THIS^.testLsbIsNotEqualTo(
	valueToTest := THIS^.LSB_ONLY,
	unexpectedValue := TRUE
);	
THIS^.testLsbIsNotEqualTo(
	valueToTest := THIS^.LSB_ONLY,
	unexpectedValue := FALSE
);
THIS^.testLsbIsNotEqualTo(
	valueToTest := THIS^.MSB_ONLY,
	unexpectedValue := TRUE
);	
THIS^.testLsbIsNotEqualTo(
	valueToTest := THIS^.MSB_ONLY,
	unexpectedValue := FALSE
);

TcUnit.TEST_FINISHED();
END_METHOD

(*

simple summary
==================
This test method tests ``assert.bitNumber.simple.lsbIsSet``
of CNM_AssertionInterfaces library with various inputs

.. <legal notes>

legal notes
=================
| SPDX-FileCopyrightText: © 2022 ekvip automation GmbH <info@ekvip.de>
| SPDX-License-Identifier: Apache-2.0
| For details check: Apache-2.0_

.. _Apache-2.0: https://www.apache.org/licenses/LICENSE-2.0

.. </legal notes>

*)

METHOD runLsbIsSetTests
VAR
	(* it's just part of the test data *)
	valueToTest	:WORD;
	(* multiplier to get various bit patterns *)
	multiplier	:UINT;
END_VAR
RETURN (NOT TcUnit.TEST_ORDERED(THIS^.getTestNameFor('lsbIsSet')));

FOR multiplier := THIS^.FIRST_MULTIPLIER TO THIS^.LAST_MULTIPLIER DO
	valueToTest := (THIS^.MULTIPLICAND * multiplier);
	THIS^.testLsbIsSet(
		valueToTest := valueToTest
	);
END_FOR

THIS^.testLsbIsSet(
	valueToTest := THIS^.MSB_ONLY
);	
THIS^.testLsbIsSet(
	valueToTest := THIS^.MSB_ONLY
);

TcUnit.TEST_FINISHED();
END_METHOD

(*

simple summary
==================
This test method tests ``assert.bitNumber.simple.lsbIsUnset``
of CNM_AssertionInterfaces library with various inputs

.. <legal notes>

legal notes
=================
| SPDX-FileCopyrightText: © 2022 ekvip automation GmbH <info@ekvip.de>
| SPDX-License-Identifier: Apache-2.0
| For details check: Apache-2.0_

.. _Apache-2.0: https://www.apache.org/licenses/LICENSE-2.0

.. </legal notes>

*)

METHOD runLsbIsUnsetTests
VAR
	(* it's just part of the test data *)
	valueToTest	:WORD;
	(* multiplier to get various bit patterns *)
	multiplier	:UINT;
END_VAR
RETURN (NOT TcUnit.TEST_ORDERED(THIS^.getTestNameFor('lsbIsUnset')));

FOR multiplier := THIS^.FIRST_MULTIPLIER TO THIS^.LAST_MULTIPLIER DO
	valueToTest := (THIS^.MULTIPLICAND * multiplier);
	THIS^.testLsbIsUnset(
		valueToTest := valueToTest
	);
END_FOR

THIS^.testLsbIsUnset(
	valueToTest := THIS^.LSB_ONLY
);	
THIS^.testLsbIsUnset(
	valueToTest := THIS^.MSB_ONLY
);

TcUnit.TEST_FINISHED();
END_METHOD

(*

simple summary
==================
This test method tests ``assert.bitNumber.simple.msbIsEqualTo``
method of CNM_AssertionInterfaces library with various inputs

.. <legal notes>

legal notes
=================
| SPDX-FileCopyrightText: © 2022 ekvip automation GmbH <info@ekvip.de>
| SPDX-License-Identifier: Apache-2.0
| For details check: Apache-2.0_

.. _Apache-2.0: https://www.apache.org/licenses/LICENSE-2.0

.. </legal notes>

*)

METHOD runMsbIsEqualToTests
VAR
	(* it's just part of the test data *)
	valueToTest	:WORD;
	(* multiplier to get various bit patterns *)
	multiplier	:UINT;
END_VAR
VAR CONSTANT
	(* number how many times the product will be rotated right *)
	NUMBER_OF_RORS :UINT := 1;
	(* multiplicand for the ``multiplier`` *)
	MULTIPLICAND :UINT := 17;
	(* first of all multipliers the test iterates *)
	FIRST_MULTIPLIER :UINT := 0;
	(* first of all multipliers the test iterates *)
	LAST_MULTIPLIER :UINT := 15;
END_VAR
RETURN (NOT TcUnit.TEST_ORDERED(THIS^.getTestNameFor('msbIsEqualTo')));

FOR multiplier := THIS^.FIRST_MULTIPLIER TO THIS^.LAST_MULTIPLIER DO
	valueToTest := ROR(THIS^.MULTIPLICAND * multiplier, THIS^.NUMBER_OF_RORS);

	THIS^.testMsbIsEqualTo(
		valueToTest := valueToTest,
		expectedValue := TRUE
	);	
	THIS^.testMsbIsEqualTo(
		valueToTest := valueToTest,
		expectedValue := FALSE
	);
END_FOR

THIS^.testMsbIsEqualTo(
	valueToTest := THIS^.LSB_ONLY,
	expectedValue := TRUE
);	
THIS^.testMsbIsEqualTo(
	valueToTest := THIS^.LSB_ONLY,
	expectedValue := FALSE
);
THIS^.testMsbIsEqualTo(
	valueToTest := THIS^.MSB_ONLY,
	expectedValue := TRUE
);	
THIS^.testMsbIsEqualTo(
	valueToTest := THIS^.MSB_ONLY,
	expectedValue := FALSE
);

TcUnit.TEST_FINISHED();
END_METHOD

(*

simple summary
==================
This test method tests ``assert.bitNumber.simple.msbIsNotEqualTo``
method of CNM_AssertionInterfaces library with various inputs

.. <legal notes>

legal notes
=================
| SPDX-FileCopyrightText: © 2022 ekvip automation GmbH <info@ekvip.de>
| SPDX-License-Identifier: Apache-2.0
| For details check: Apache-2.0_

.. _Apache-2.0: https://www.apache.org/licenses/LICENSE-2.0

.. </legal notes>

*)

METHOD runMsbIsNotEqualToTests
VAR
	(* it's just part of the test data *)
	valueToTest	:WORD;
	(* multiplier to get various bit patterns *)
	multiplier	:UINT;
END_VAR
RETURN (NOT TcUnit.TEST_ORDERED(THIS^.getTestNameFor('msbIsNotEqualTo')));

FOR multiplier := THIS^.FIRST_MULTIPLIER TO THIS^.LAST_MULTIPLIER DO
	valueToTest := ROR(THIS^.MULTIPLICAND * multiplier, THIS^.NUMBER_OF_RORS);
	THIS^.testMsbIsNotEqualTo(
		valueToTest := valueToTest,
		unexpectedValue := TRUE
	);	
	THIS^.testMsbIsNotEqualTo(
		valueToTest := valueToTest,
		unexpectedValue := FALSE
	);
END_FOR

THIS^.testMsbIsNotEqualTo(
	valueToTest := THIS^.LSB_ONLY,
	unexpectedValue := TRUE
);	
THIS^.testMsbIsNotEqualTo(
	valueToTest := THIS^.LSB_ONLY,
	unexpectedValue := FALSE
);
THIS^.testMsbIsNotEqualTo(
	valueToTest := THIS^.MSB_ONLY,
	unexpectedValue := TRUE
);	
THIS^.testMsbIsNotEqualTo(
	valueToTest := THIS^.MSB_ONLY,
	unexpectedValue := FALSE
);

TcUnit.TEST_FINISHED();
END_METHOD

(*

simple summary
==================
This test method tests ``assert.bitNumber.simple.msbIsSet``
of CNM_AssertionInterfaces library with various inputs

.. <legal notes>

legal notes
=================
| SPDX-FileCopyrightText: © 2022 ekvip automation GmbH <info@ekvip.de>
| SPDX-License-Identifier: Apache-2.0
| For details check: Apache-2.0_

.. _Apache-2.0: https://www.apache.org/licenses/LICENSE-2.0

.. </legal notes>

*)

METHOD runMsbIsSetTests
VAR
	(* it's just part of the test data *)
	valueToTest	:WORD;
	(* multiplier to get various bit patterns *)
	multiplier	:UINT;
END_VAR
RETURN (NOT TcUnit.TEST_ORDERED(THIS^.getTestNameFor('msbIsUnset')));

FOR multiplier := THIS^.FIRST_MULTIPLIER TO THIS^.LAST_MULTIPLIER DO
	valueToTest := ROR(THIS^.MULTIPLICAND * multiplier, THIS^.NUMBER_OF_RORS);
	THIS^.testMsbIsSet(
		valueToTest := valueToTest
	);
END_FOR

THIS^.testMsbIsSet(
	valueToTest := THIS^.LSB_ONLY
);	
THIS^.testMsbIsSet(
	valueToTest := THIS^.MSB_ONLY
);

TcUnit.TEST_FINISHED();
END_METHOD

(*

simple summary
==================
This test method tests ``assert.bitNumber.simple.msbIsUnset``
of CNM_AssertionInterfaces library with various inputs

.. <legal notes>

legal notes
=================
| SPDX-FileCopyrightText: © 2022 ekvip automation GmbH <info@ekvip.de>
| SPDX-License-Identifier: Apache-2.0
| For details check: Apache-2.0_

.. _Apache-2.0: https://www.apache.org/licenses/LICENSE-2.0

.. </legal notes>

*)

METHOD runMsbIsUnsetTests
VAR
	(* it's just part of the test data *)
	valueToTest	:WORD;
	(* multiplier to get various bit patterns *)
	multiplier	:UINT;
END_VAR
RETURN (NOT TcUnit.TEST_ORDERED(THIS^.getTestNameFor('msbIsSet')));

FOR multiplier := THIS^.FIRST_MULTIPLIER TO THIS^.LAST_MULTIPLIER DO
	valueToTest := ROR(THIS^.MULTIPLICAND * multiplier, THIS^.NUMBER_OF_RORS);
	THIS^.testMsbIsSet(
		valueToTest := valueToTest
	);
END_FOR

THIS^.testMsbIsSet(
	valueToTest := THIS^.LSB_ONLY
);	
THIS^.testMsbIsSet(
	valueToTest := THIS^.MSB_ONLY
);

TcUnit.TEST_FINISHED();
END_METHOD

(*

simple summary
==================
This test method tests ``assert.bitNumber.simple.orMaskIsEqualTo``
method of CNM_AssertionInterfaces library with various inputs

.. <legal notes>

legal notes
=================
| SPDX-FileCopyrightText: © 2022 ekvip automation GmbH <info@ekvip.de>
| SPDX-License-Identifier: Apache-2.0
| For details check: Apache-2.0_

.. _Apache-2.0: https://www.apache.org/licenses/LICENSE-2.0

.. </legal notes>

*)

METHOD runOrMaskIsEqualToTests
VAR
	(* shift to iterate through the bit numbers *)
	shift				:UINT;
	(* it's just part of the test data *)
	valueToTest		:WORD;
	(* mask with the bit iteration *)
	mask				:WORD;
END_VAR
RETURN (NOT TcUnit.TEST_ORDERED(THIS^.getTestNameFor('orMaskIsEqualTo')));

FOR shift:= THIS^.FIRST_BIT TO THIS^.LAST_BIT DO
	mask := SHL(THIS^.LSB_ONLY, shift);
	valueToTest := SHR(THIS^.MSB_ONLY, shift);
	THIS^.testOrMaskIsEqualTo(
		valueToTest := valueToTest,
		mask  := mask,
		expected := (mask OR valueToTest)
	);
	THIS^.testOrMaskIsEqualTo(
		valueToTest := valueToTest,
		mask  := mask,
		expected := (NOT (mask OR valueToTest))
	);
	THIS^.testAndMaskIsEqualTo(
		valueToTest := mask,
		mask  := (NOT mask),
		expected := THIS^.NO_BIT_SET
	);
	THIS^.testAndMaskIsEqualTo(
		valueToTest := mask,
		mask  := (NOT mask),
		expected := THIS^.ALL_BITS_SET
	);	
END_FOR

THIS^.testAndMaskIsEqualTo(
	valueToTest := THIS^.NO_BIT_SET,
	mask  := THIS^.NO_BIT_SET,
	expected := THIS^.NO_BIT_SET
);
THIS^.testAndMaskIsEqualTo(
	valueToTest := THIS^.NO_BIT_SET,
	mask  := THIS^.NO_BIT_SET,
	expected := THIS^.ALL_BITS_SET
);	

THIS^.testAndMaskIsEqualTo(
	valueToTest := THIS^.ALL_BITS_SET,
	mask  := THIS^.ALL_BITS_SET,
	expected := THIS^.ALL_BITS_SET
);
THIS^.testAndMaskIsEqualTo(
	valueToTest := THIS^.ALL_BITS_SET,
	mask  := THIS^.ALL_BITS_SET,
	expected := THIS^.NO_BIT_SET
);	

TcUnit.TEST_FINISHED();
END_METHOD

(*

simple summary
==================
This test method tests ``assert.bitNumber.simple.orMaskIsNotEqualTo``
method of CNM_AssertionInterfaces library with various inputs

.. <legal notes>

legal notes
=================
| SPDX-FileCopyrightText: © 2022 ekvip automation GmbH <info@ekvip.de>
| SPDX-License-Identifier: Apache-2.0
| For details check: Apache-2.0_

.. _Apache-2.0: https://www.apache.org/licenses/LICENSE-2.0

.. </legal notes>

*)

METHOD runOrMaskIsNotEqualToTests
VAR
	(* shift to iterate through the bit numbers *)
	shift				:UINT;
	(* it's just part of the test data *)
	valueToTest		:WORD;
	(* mask with the bit iteration *)
	mask				:WORD;
END_VAR
RETURN (NOT TcUnit.TEST_ORDERED(THIS^.getTestNameFor('orMaskIsNotEqualTo')));

FOR shift:= THIS^.FIRST_BIT TO THIS^.LAST_BIT DO
	mask := SHL(THIS^.LSB_ONLY, shift);
	valueToTest := SHR(THIS^.MSB_ONLY, shift);
	THIS^.testOrMaskIsNotEqualTo(
		valueToTest := valueToTest,
		mask  := mask,
		unexpected := (mask OR valueToTest)
	);
	THIS^.testOrMaskIsNotEqualTo(
		valueToTest := valueToTest,
		mask  := mask,
		unexpected := (NOT (mask OR valueToTest))
	);
	THIS^.testOrMaskIsNotEqualTo(
		valueToTest := mask,
		mask  := (NOT mask),
		unexpected := THIS^.NO_BIT_SET
	);
	THIS^.testOrMaskIsNotEqualTo(
		valueToTest := mask,
		mask  := (NOT mask),
		unexpected := THIS^.ALL_BITS_SET
	);	
END_FOR

THIS^.testOrMaskIsNotEqualTo(
	valueToTest := THIS^.NO_BIT_SET,
	mask  := THIS^.NO_BIT_SET,
	unexpected := THIS^.NO_BIT_SET
);
THIS^.testOrMaskIsNotEqualTo(
	valueToTest := THIS^.NO_BIT_SET,
	mask  := THIS^.NO_BIT_SET,
	unexpected := THIS^.ALL_BITS_SET
);	

THIS^.testOrMaskIsNotEqualTo(
	valueToTest := THIS^.ALL_BITS_SET,
	mask  := THIS^.ALL_BITS_SET,
	unexpected := THIS^.ALL_BITS_SET
);
THIS^.testOrMaskIsNotEqualTo(
	valueToTest := THIS^.ALL_BITS_SET,
	mask  := THIS^.ALL_BITS_SET,
	unexpected := THIS^.NO_BIT_SET
);	

TcUnit.TEST_FINISHED();
END_METHOD

(*

simple summary
==================
This test method tests ``assert.bitNumber.simple.valueIsEqualTo``
method of CNM_AssertionInterfaces library with various inputs

.. <legal notes>

legal notes
=================
| SPDX-FileCopyrightText: © 2022 ekvip automation GmbH <info@ekvip.de>
| SPDX-License-Identifier: Apache-2.0
| For details check: Apache-2.0_

.. _Apache-2.0: https://www.apache.org/licenses/LICENSE-2.0

.. </legal notes>

*)

METHOD runValueIsEqualToTests
RETURN (NOT TcUnit.TEST_ORDERED(THIS^.getTestNameFor('valueIsEqualTo')));

THIS^.testValueIsEqualTo(
	valueToTest := THIS^.NO_BIT_SET,
	expected := THIS^.ALL_BITS_SET
);
THIS^.testValueIsEqualTo(
	valueToTest := THIS^.NO_BIT_SET,
	expected := THIS^.NO_BIT_SET
);
THIS^.testValueIsEqualTo(
	valueToTest := THIS^.ALL_BITS_SET,
	expected := THIS^.ALL_BITS_SET
);
THIS^.testValueIsEqualTo(
	valueToTest := THIS^.ALL_BITS_SET,
	expected := THIS^.NO_BIT_SET
);
THIS^.testValueIsEqualTo(
	valueToTest := THIS^.LSB_ONLY,
	expected := THIS^.LSB_ONLY
);
THIS^.testValueIsEqualTo(
	valueToTest := THIS^.LSB_ONLY,
	expected := THIS^.MSB_ONLY
);
THIS^.testValueIsEqualTo(
	valueToTest := THIS^.MSB_ONLY,
	expected := THIS^.MSB_ONLY
);
THIS^.testValueIsEqualTo(
	valueToTest := THIS^.MSB_ONLY,
	expected := THIS^.LSB_ONLY
);

TcUnit.TEST_FINISHED();
END_METHOD

(*

simple summary
==================
This test method tests ``assert.bitNumber.simple.valueIsGreaterThan``
method of CNM_AssertionInterfaces library with various inputs

.. <legal notes>

legal notes
=================
| SPDX-FileCopyrightText: © 2022 ekvip automation GmbH <info@ekvip.de>
| SPDX-License-Identifier: Apache-2.0
| For details check: Apache-2.0_

.. _Apache-2.0: https://www.apache.org/licenses/LICENSE-2.0

.. </legal notes>

*)

METHOD runValueIsGreaterTests
RETURN (NOT TcUnit.TEST_ORDERED(THIS^.getTestNameFor('valueIsGreaterThan')));

THIS^.testValueIsGreater(
	valueToTest := THIS^.NO_BIT_SET,
	less := THIS^.ALL_BITS_SET
);
THIS^.testValueIsGreater(
	valueToTest := THIS^.NO_BIT_SET,
	less := THIS^.NO_BIT_SET
);
THIS^.testValueIsGreater(
	valueToTest := THIS^.ALL_BITS_SET,
	less := THIS^.ALL_BITS_SET
);
THIS^.testValueIsGreater(
	valueToTest := THIS^.ALL_BITS_SET,
	less := THIS^.NO_BIT_SET
);
THIS^.testValueIsGreater(
	valueToTest := THIS^.LSB_ONLY,
	less := THIS^.LSB_ONLY
);
THIS^.testValueIsGreater(
	valueToTest := THIS^.LSB_ONLY,
	less := THIS^.NO_BIT_SET
);
THIS^.testValueIsGreater(
	valueToTest := THIS^.LSB_ONLY,
	less := (THIS^.LSB_ONLY+THIS^.LSB_ONLY)
);
THIS^.testValueIsGreater(
	valueToTest := THIS^.MSB_ONLY,
	less := THIS^.MSB_ONLY
);
THIS^.testValueIsGreater(
	valueToTest := THIS^.MSB_ONLY,
	less := (NOT THIS^.MSB_ONLY)
);
THIS^.testValueIsGreater(
	valueToTest := THIS^.MSB_ONLY,
	less := THIS^.ALL_BITS_SET
);
TcUnit.TEST_FINISHED();
END_METHOD

(*

simple summary
==================
This test method tests ``assert.bitNumber.simple.valueIsInRangeOf``
method of CNM_AssertionInterfaces library with various inputs

.. <legal notes>

legal notes
=================
| SPDX-FileCopyrightText: © 2022 ekvip automation GmbH <info@ekvip.de>
| SPDX-License-Identifier: Apache-2.0
| For details check: Apache-2.0_

.. _Apache-2.0: https://www.apache.org/licenses/LICENSE-2.0

.. </legal notes>

*)

METHOD runValueIsInRangeOfTests
RETURN (NOT TcUnit.TEST_ORDERED(THIS^.getTestNameFor('valueIsInRangeOf')));

THIS^.testValueIsInRangeOf(
	lower := THIS^.NO_BIT_SET,
	valueToTest := THIS^.LSB_ONLY,
	upper := THIS^.ALL_BITS_SET
);
THIS^.testValueIsInRangeOf(
	lower := THIS^.NO_BIT_SET,
	valueToTest := THIS^.NO_BIT_SET,
	upper := THIS^.NO_BIT_SET
);
THIS^.testValueIsInRangeOf(
	lower := THIS^.ALL_BITS_SET,
	valueToTest := THIS^.ALL_BITS_SET,
	upper := THIS^.ALL_BITS_SET
);
THIS^.testValueIsInRangeOf(
	lower := THIS^.ALL_BITS_SET,
	valueToTest := THIS^.LSB_ONLY,
	upper := THIS^.NO_BIT_SET
);
THIS^.testValueIsInRangeOf(
	lower := THIS^.ALL_BITS_SET,
	valueToTest := THIS^.NO_BIT_SET,
	upper := THIS^.NO_BIT_SET
);

TEST_FINISHED();
END_METHOD

(*

simple summary
==================
This test method tests ``assert.bitNumber.simple.valueIsLessThan``
method of CNM_AssertionInterfaces library with various inputs

.. <legal notes>

legal notes
=================
| SPDX-FileCopyrightText: © 2022 ekvip automation GmbH <info@ekvip.de>
| SPDX-License-Identifier: Apache-2.0
| For details check: Apache-2.0_

.. _Apache-2.0: https://www.apache.org/licenses/LICENSE-2.0

.. </legal notes>

*)

METHOD runValueIsLessThanTests
RETURN (NOT TcUnit.TEST_ORDERED(THIS^.getTestNameFor('valueIsLessThan')));

THIS^.testValueIsLessThan(
	valueToTest := THIS^.NO_BIT_SET,
	greater := THIS^.ALL_BITS_SET
);
THIS^.testValueIsLessThan(
	valueToTest := THIS^.NO_BIT_SET,
	greater := THIS^.NO_BIT_SET
);
THIS^.testValueIsLessThan(
	valueToTest := THIS^.ALL_BITS_SET,
	greater := THIS^.ALL_BITS_SET
);
THIS^.testValueIsLessThan(
	valueToTest := THIS^.ALL_BITS_SET,
	greater := THIS^.NO_BIT_SET
);
THIS^.testValueIsLessThan(
	valueToTest := THIS^.LSB_ONLY,
	greater := THIS^.LSB_ONLY
);
THIS^.testValueIsLessThan(
	valueToTest := THIS^.LSB_ONLY,
	greater := THIS^.NO_BIT_SET
);
THIS^.testValueIsLessThan(
	valueToTest := THIS^.MSB_ONLY,
	greater := (THIS^.MSB_ONLY+THIS^.LSB_ONLY)
);
THIS^.testValueIsLessThan(
	valueToTest := THIS^.MSB_ONLY,
	greater := THIS^.MSB_ONLY
);
THIS^.testValueIsLessThan(
	valueToTest := THIS^.MSB_ONLY,
	greater := (NOT THIS^.MSB_ONLY)
);
THIS^.testValueIsLessThan(
	valueToTest := THIS^.MSB_ONLY,
	greater := THIS^.ALL_BITS_SET
);

TcUnit.TEST_FINISHED();
END_METHOD

(*

simple summary
==================
This test method tests ``assert.bitNumber.simple.valueIsMax``
method of CNM_AssertionInterfaces library with various inputs

.. <legal notes>

legal notes
=================
| SPDX-FileCopyrightText: © 2022 ekvip automation GmbH <info@ekvip.de>
| SPDX-License-Identifier: Apache-2.0
| For details check: Apache-2.0_

.. _Apache-2.0: https://www.apache.org/licenses/LICENSE-2.0

.. </legal notes>

*)

METHOD runValueIsMaxTests
RETURN (NOT TcUnit.TEST_ORDERED(THIS^.getTestNameFor('valueIsMax')));

THIS^.testValueIsMax(
	valueToTest := THIS^.NO_BIT_SET,
	maximum := THIS^.LSB_ONLY
);
THIS^.testValueIsMax(
	valueToTest := THIS^.LSB_ONLY,
	maximum := THIS^.NO_BIT_SET
);
THIS^.testValueIsMax(
	valueToTest := THIS^.NO_BIT_SET,
	maximum := THIS^.NO_BIT_SET
);
THIS^.testValueIsMax(
	valueToTest := THIS^.ALL_BITS_SET,
	maximum := ALL_BITS_SET
);
THIS^.testValueIsMax(
	valueToTest := (THIS^.ALL_BITS_SET-THIS^.LSB_ONLY),
	maximum := THIS^.ALL_BITS_SET
);
THIS^.testValueIsMax(
	valueToTest := THIS^.ALL_BITS_SET,
	maximum := (THIS^.ALL_BITS_SET-THIS^.LSB_ONLY)
);
THIS^.testValueIsMax(
	valueToTest := THIS^.MSB_ONLY,
	maximum := (THIS^.MSB_ONLY+THIS^.LSB_ONLY)
);
THIS^.testValueIsMax(
	valueToTest := (THIS^.MSB_ONLY+THIS^.LSB_ONLY),
	maximum := THIS^.MSB_ONLY
);
THIS^.testValueIsMax(
	valueToTest := THIS^.MSB_ONLY,
	maximum := (NOT THIS^.MSB_ONLY)
);
THIS^.testValueIsMax(
	valueToTest := (NOT THIS^.MSB_ONLY),
	maximum := THIS^.MSB_ONLY
);
THIS^.testValueIsMax(
	valueToTest := THIS^.MSB_ONLY,
	maximum := THIS^.MSB_ONLY
);

TcUnit.TEST_FINISHED();
END_METHOD

(*

simple summary
==================
This test method tests ``assert.bitNumber.simple.valueIsMin``
method of CNM_AssertionInterfaces library with various inputs

.. <legal notes>

legal notes
=================
| SPDX-FileCopyrightText: © 2022 ekvip automation GmbH <info@ekvip.de>
| SPDX-License-Identifier: Apache-2.0
| For details check: Apache-2.0_

.. _Apache-2.0: https://www.apache.org/licenses/LICENSE-2.0

.. </legal notes>

*)

METHOD runValueIsMinTests
RETURN (NOT TcUnit.TEST_ORDERED(THIS^.getTestNameFor('valueIsMin')));

THIS^.testValueIsMin(
	valueToTest := THIS^.NO_BIT_SET,
	minimum := THIS^.LSB_ONLY
);
THIS^.testValueIsMin(
	valueToTest := THIS^.LSB_ONLY,
	minimum := THIS^.NO_BIT_SET
);
THIS^.testValueIsMin(
	valueToTest := THIS^.NO_BIT_SET,
	minimum := THIS^.NO_BIT_SET
);
THIS^.testValueIsMin(
	valueToTest := THIS^.ALL_BITS_SET,
	minimum := ALL_BITS_SET
);
THIS^.testValueIsMin(
	valueToTest := (THIS^.ALL_BITS_SET-THIS^.LSB_ONLY),
	minimum := THIS^.ALL_BITS_SET
);
THIS^.testValueIsMin(
	valueToTest := THIS^.ALL_BITS_SET,
	minimum := (THIS^.ALL_BITS_SET-THIS^.LSB_ONLY)
);
THIS^.testValueIsMin(
	valueToTest := THIS^.MSB_ONLY,
	minimum := (THIS^.MSB_ONLY+THIS^.LSB_ONLY)
);
THIS^.testValueIsMin(
	valueToTest := (THIS^.MSB_ONLY+THIS^.LSB_ONLY),
	minimum := THIS^.MSB_ONLY
);
THIS^.testValueIsMin(
	valueToTest := THIS^.MSB_ONLY,
	minimum := (NOT THIS^.MSB_ONLY)
);
THIS^.testValueIsMin(
	valueToTest := (NOT THIS^.MSB_ONLY),
	minimum := THIS^.MSB_ONLY
);
THIS^.testValueIsMin(
	valueToTest := THIS^.MSB_ONLY,
	minimum := THIS^.MSB_ONLY
);

TcUnit.TEST_FINISHED();
END_METHOD

(*

simple summary
==================
This test method tests ``assert.bitNumber.simple.valueIsNotEqualTo``
method of CNM_AssertionInterfaces library with various inputs

.. <legal notes>

legal notes
=================
| SPDX-FileCopyrightText: © 2022 ekvip automation GmbH <info@ekvip.de>
| SPDX-License-Identifier: Apache-2.0
| For details check: Apache-2.0_

.. _Apache-2.0: https://www.apache.org/licenses/LICENSE-2.0

.. </legal notes>

*)

METHOD runValueIsNotEqualToTests
RETURN (NOT TcUnit.TEST_ORDERED(THIS^.getTestNameFor('valueIsNotEqualTo')));

THIS^.testValueIsNotEqualTo(
	valueToTest := THIS^.NO_BIT_SET,
	unexpected := THIS^.ALL_BITS_SET
);
THIS^.testValueIsNotEqualTo(
	valueToTest := THIS^.NO_BIT_SET,
	unexpected := THIS^.NO_BIT_SET
);
THIS^.testValueIsNotEqualTo(
	valueToTest := THIS^.ALL_BITS_SET,
	unexpected := THIS^.ALL_BITS_SET
);
THIS^.testValueIsNotEqualTo(
	valueToTest := THIS^.ALL_BITS_SET,
	unexpected := THIS^.NO_BIT_SET
);
THIS^.testValueIsNotEqualTo(
	valueToTest := THIS^.LSB_ONLY,
	unexpected := THIS^.LSB_ONLY
);
THIS^.testValueIsNotEqualTo(
	valueToTest := THIS^.LSB_ONLY,
	unexpected := THIS^.MSB_ONLY
);
THIS^.testValueIsNotEqualTo(
	valueToTest := THIS^.MSB_ONLY,
	unexpected := THIS^.MSB_ONLY
);
THIS^.testValueIsNotEqualTo(
	valueToTest := THIS^.MSB_ONLY,
	unexpected := THIS^.LSB_ONLY
);

TcUnit.TEST_FINISHED();
END_METHOD

(*

simple summary
==================
This test method tests ``assert.bitNumber.simple.xorMaskIsEqualTo``
method of CNM_AssertionInterfaces library with various inputs

.. <legal notes>

legal notes
=================
| SPDX-FileCopyrightText: © 2022 ekvip automation GmbH <info@ekvip.de>
| SPDX-License-Identifier: Apache-2.0
| For details check: Apache-2.0_

.. _Apache-2.0: https://www.apache.org/licenses/LICENSE-2.0

.. </legal notes>

*)

METHOD runXorMaskIsEqualToTests
VAR
	(* shift to iterate through the bit numbers *)
	shift				:UINT;
	(* it's just part of the test data *)
	valueToTest		:WORD;
	(* mask with the bit iteration *)
	mask				:WORD;
END_VAR
RETURN (NOT TcUnit.TEST_ORDERED(THIS^.getTestNameFor('xorMaskIsEqualTo')));

FOR shift:= THIS^.FIRST_BIT TO THIS^.LAST_BIT DO
	mask := SHL(THIS^.LSB_ONLY, shift);
	valueToTest := (NOT mask);
	THIS^.testOrMaskIsEqualTo(
		valueToTest := valueToTest,
		mask  := mask,
		expected := THIS^.ALL_BITS_SET
	);
	THIS^.testOrMaskIsEqualTo(
		valueToTest := valueToTest,
		mask  := mask,
		expected := THIS^.NO_BIT_SET
	);
	THIS^.testAndMaskIsEqualTo(
		valueToTest := mask,
		mask  := mask,
		expected := THIS^.NO_BIT_SET
	);
	THIS^.testAndMaskIsEqualTo(
		valueToTest := mask,
		mask  := mask,
		expected := mask
	);	
END_FOR

THIS^.testAndMaskIsEqualTo(
	valueToTest := THIS^.NO_BIT_SET,
	mask  := THIS^.NO_BIT_SET,
	expected := THIS^.NO_BIT_SET
);
THIS^.testAndMaskIsEqualTo(
	valueToTest := THIS^.NO_BIT_SET,
	mask  := THIS^.NO_BIT_SET,
	expected := THIS^.ALL_BITS_SET
);	

THIS^.testAndMaskIsEqualTo(
	valueToTest := THIS^.ALL_BITS_SET,
	mask  := THIS^.ALL_BITS_SET,
	expected := THIS^.ALL_BITS_SET
);
THIS^.testAndMaskIsEqualTo(
	valueToTest := THIS^.ALL_BITS_SET,
	mask  := THIS^.ALL_BITS_SET,
	expected := THIS^.NO_BIT_SET
);	

TcUnit.TEST_FINISHED();
END_METHOD

(*

simple summary
==================
This test method tests ``assert.bitNumber.simple.xorMaskIsNotEqualTo``
method of CNM_AssertionInterfaces library with various inputs

.. <legal notes>

legal notes
=================
| SPDX-FileCopyrightText: © 2022 ekvip automation GmbH <info@ekvip.de>
| SPDX-License-Identifier: Apache-2.0
| For details check: Apache-2.0_

.. _Apache-2.0: https://www.apache.org/licenses/LICENSE-2.0

.. </legal notes>

*)

METHOD runXorMaskIsNotEqualToTests
VAR
	(* shift to iterate through the bit numbers *)
	shift				:UINT;
	(* it's just part of the test data *)
	valueToTest			:WORD;
	(* mask with the bit iteration *)
	mask				:WORD;
END_VAR
RETURN (NOT TcUnit.TEST_ORDERED(THIS^.getTestNameFor('xorMaskIsNotEqualTo')));

FOR shift:= THIS^.FIRST_BIT TO THIS^.LAST_BIT DO
	mask := SHL(THIS^.LSB_ONLY, shift);
	valueToTest := (NOT mask);
	THIS^.testXorMaskIsNotEqualTo(
		valueToTest := valueToTest,
		mask  := mask,
		unexpected := THIS^.ALL_BITS_SET
	);
	THIS^.testXorMaskIsNotEqualTo(
		valueToTest := valueToTest,
		mask  := mask,
		unexpected := THIS^.NO_BIT_SET
	);
	THIS^.testXorMaskIsNotEqualTo(
		valueToTest := mask,
		mask  := mask,
		unexpected := THIS^.NO_BIT_SET
	);
	THIS^.testXorMaskIsNotEqualTo(
		valueToTest := mask,
		mask  := mask,
		unexpected := mask
	);	
END_FOR

THIS^.testXorMaskIsNotEqualTo(
	valueToTest := THIS^.NO_BIT_SET,
	mask  := THIS^.NO_BIT_SET,
	unexpected := THIS^.NO_BIT_SET
);
THIS^.testXorMaskIsNotEqualTo(
	valueToTest := THIS^.NO_BIT_SET,
	mask  := THIS^.NO_BIT_SET,
	unexpected := THIS^.ALL_BITS_SET
);	

THIS^.testXorMaskIsNotEqualTo(
	valueToTest := THIS^.ALL_BITS_SET,
	mask  := THIS^.ALL_BITS_SET,
	unexpected := THIS^.ALL_BITS_SET
);
THIS^.testXorMaskIsNotEqualTo(
	valueToTest := THIS^.ALL_BITS_SET,
	mask  := THIS^.ALL_BITS_SET,
	unexpected := THIS^.NO_BIT_SET
);	

THIS^.testXorMaskIsNotEqualTo(
	valueToTest := THIS^.ALL_BITS_SET,
	mask  := THIS^.NO_BIT_SET,
	unexpected := THIS^.ALL_BITS_SET
);
THIS^.testXorMaskIsNotEqualTo(
	valueToTest := THIS^.ALL_BITS_SET,
	mask  := THIS^.NO_BIT_SET,
	unexpected := THIS^.NO_BIT_SET
);

TcUnit.TEST_FINISHED();
END_METHOD

(*

simple summary
==================
This test method tests ``assert.bitNumber.simple.andMaskIsEqualTo``
method of CNM_AssertionInterfaces library, 
it provides the possibility to handover test data via parameter 


.. <legal notes>

legal notes
=================
| SPDX-FileCopyrightText: © 2022 ekvip automation GmbH <info@ekvip.de>
| SPDX-License-Identifier: Apache-2.0
| For details check: Apache-2.0_

.. _Apache-2.0: https://www.apache.org/licenses/LICENSE-2.0

.. </legal notes>

parameters
==========

*)

METHOD testAndMaskIsEqualTo 
VAR_INPUT
	(* for the test it's the parameter ``currentValue`` *)
	valueToTest	:WORD;
	(* it's the mask for the currentValue *)
	mask		:WORD;
	(* for the test it's the parameter ``expectedValue`` *)
	expected	:WORD;
END_VAR
VAR
	(* just the expectation if the assertion to test must be worng or true *)
	assertionIsWrong		:BOOL;
	(* result of the bit operation to determine the value of ``assertionIsWrong`` *)
	result					:WORD;
	(* contains the format string for the test message *)
	message					:Tc2_System.T_MaxString;
	(* TwinCAT printf with the test message *)
	messageStringBuilder	:Tc2_Utilities.FB_FormatString;
END_VAR
THIS^.assertorContainer.resetAssertor();

result := (valueToTest AND mask);
assertionIsWrong := (result <> expected);
message := SEL(
	assertionIsWrong,
	'currentValue: 16#%.4X AND mask: 16#%.4X is 16#%.4X expectedValue: 16#%.4X assertion must be TRUE', 
	'currentValue: 16#%.4X AND mask: 16#%.4X is 16#%.4X expectedValue: 16#%.4X assertion must be FALSE'
);
messageStringBuilder(
	sFormat := message,
	arg1 := THIS^.AnyToArg(valueToTest),
	arg2 := THIS^.AnyToArg(mask),
	arg3 := THIS^.AnyToArg(result),
	arg4 := THIS^.AnyToArg(expected)
);

THIS^.assertorContainer.assertor.assert.bitNumber.simple.andMaskIsEqualTo(
	currentValue	:= valueToTest,
	mask 			:= mask,
	expectedValue	:= expected,
	message			:= ''
);

THIS^.AssertEquals_BOOL(
	Expected 	:= assertionIsWrong,
	Actual 		:= THIS^.assertorContainer.wasAssertionWrong,
	Message 	:= messageStringBuilder.sOut
);
END_METHOD

(*

simple summary
==================
This test method tests ``assert.bitNumber.simple.andMaskIsNotEqualTo``
method of CNM_AssertionInterfaces library, 
it provides the possibility to handover test data via parameter 


.. <legal notes>

legal notes
=================
| SPDX-FileCopyrightText: © 2022 ekvip automation GmbH <info@ekvip.de>
| SPDX-License-Identifier: Apache-2.0
| For details check: Apache-2.0_

.. _Apache-2.0: https://www.apache.org/licenses/LICENSE-2.0

.. </legal notes>

parameters
==========

*)

METHOD testAndMaskIsNotEqualTo 
VAR_INPUT
	(* for the test it's the parameter ``currentValue`` *)
	valueToTest	:WORD;
	(* it's the mask for the currentValue *)
	mask		:WORD;
	(* for the test it's the parameter ``unexpectedValue`` *)
	unexpected	:WORD;
END_VAR
VAR
	(* just the expectation if the assertion to test must be worng or true *)
	assertionIsWrong		:BOOL;
	(* result of the bit operation to determine the value of ``assertionIsWrong`` *)
	result					:WORD;
	(* contains the format string for the test message *)
	message					:Tc2_System.T_MaxString;
	(* TwinCAT printf with the test message *)
	messageStringBuilder	:Tc2_Utilities.FB_FormatString;
END_VAR
THIS^.assertorContainer.resetAssertor();

result := (valueToTest AND mask);
assertionIsWrong := (result = unexpected);
message := SEL(
	assertionIsWrong,
	'currentValue: 16#%.4X AND mask: 16#%.4X is 16#%.4X unexpectedValue: 16#%.4X assertion must be TRUE', 
	'currentValue: 16#%.4X AND mask: 16#%.4X is 16#%.4X unexpectedValue: 16#%.4X assertion must be FLASE'
);
messageStringBuilder(
	sFormat := message,
	arg1 := THIS^.AnyToArg(valueToTest),
	arg2 := THIS^.AnyToArg(mask),
	arg3 := THIS^.AnyToArg(result),
	arg4 := THIS^.AnyToArg(unexpected)
);

THIS^.assertorContainer.assertor.assert.bitNumber.simple.andMaskIsNotEqualTo(
	currentValue	:= valueToTest,
	mask 			:= mask,
	unexpectedValue	:= unexpected,
	message			:= ''
);

THIS^.AssertEquals_BOOL(
	Expected 	:= assertionIsWrong,
	Actual 		:= THIS^.assertorContainer.wasAssertionWrong,
	Message 	:= messageStringBuilder.sOut
);
END_METHOD

(*

simple summary
==================
This test method tests ``assert.bitNumber.simple.bitXIsEqualTo``
method of CNM_AssertionInterfaces library, 
it provides the possibility to handover test data via parameter 


.. <legal notes>

legal notes
=================
| SPDX-FileCopyrightText: © 2022 ekvip automation GmbH <info@ekvip.de>
| SPDX-License-Identifier: Apache-2.0
| For details check: Apache-2.0_

.. _Apache-2.0: https://www.apache.org/licenses/LICENSE-2.0

.. </legal notes>

parameters
==========

*)

METHOD testBitXIsEqualTo
VAR_INPUT
	(* for the test it's the parameter ``currentValue`` *)
	valueToTest			:WORD;
	(* the bit number to check in this test, it's the parameter ``number``*)
	bitNumberToCheck	:CNM_AssertionInterfaces.BitNumberWord;
	(* this is the expected value of the bit ``bitNumberToCheck``, it's the parameter ``expectedValue`` *)
	bitIsSet			:BOOL;
END_VAR
VAR
	(* just the expectation if the assertion to test must be worng or true *)
	assertionIsWrong		:BOOL;
	(* bit with the number of ``bitNumberToCheck`` filtered from ``valueToTest`` *)
	specificBitOnly			:WORD;
	(* the bit number ``bitNumberToCheck`` is set to the value of ``bitIsSet`` only *)
	testBitOnly				:WORD;
	(* contains the format string for the test message *)
	message					:Tc2_System.T_MaxString;
	(* TwinCAT printf with the test message *)
	messageStringBuilder	:Tc2_Utilities.FB_FormatString;
END_VAR
THIS^.assertorContainer.resetAssertor();

specificBitOnly := (valueToTest AND SHL(THIS^.LSB_ONLY,bitNumberToCheck));
testBitOnly		:= SHL(TO_WORD(bitIsSet),bitNumberToCheck);
assertionIsWrong := (specificBitOnly <> testBitOnly);

message := 'Bit number %d in currentValue: 16#%.4X ';
message := SEL(
	(specificBitOnly > THIS^.NO_BIT_SET),
	Tc2_Standard.CONCAT(message, 'is unset '),
	Tc2_Standard.CONCAT(message, 'is set ')
);
message := SEL(
	(testBitOnly > THIS^.NO_BIT_SET),
	Tc2_Standard.CONCAT(message, 'expectedValue: is unset (FALSE) '),
	Tc2_Standard.CONCAT(message, 'expectedValue: is set (TRUE)  ')
);
message := SEL(
	assertionIsWrong,
	Tc2_Standard.CONCAT(message, 'assertion must be TRUE'),
	Tc2_Standard.CONCAT(message, 'assertion must be FALSE')
);
messageStringBuilder(
	sFormat := message,
	arg1 := THIS^.AnyToArg(bitNumberToCheck),
	arg2 := THIS^.AnyToArg(valueToTest)
);


THIS^.assertorContainer.assertor.assert.bitNumber.simple.bitXIsEqualTo(
	currentValue 	:= valueToTest,
	number			:= bitNumberToCheck,
	expectedValue	:= bitIsSet,
	message			:= ''  
); 

THIS^.AssertEquals_BOOL(
	Expected 	:= assertionIsWrong,
	Actual 		:= THIS^.assertorContainer.wasAssertionWrong,
	Message 	:= messageStringBuilder.sOut
);
END_METHOD

(*

simple summary
==================
This test method tests ``assert.bitNumber.simple.bitXIsNotEqualTo``
method of CNM_AssertionInterfaces library, 
it provides the possibility to handover test data via parameter 


.. <legal notes>

legal notes
=================
| SPDX-FileCopyrightText: © 2022 ekvip automation GmbH <info@ekvip.de>
| SPDX-License-Identifier: Apache-2.0
| For details check: Apache-2.0_

.. _Apache-2.0: https://www.apache.org/licenses/LICENSE-2.0

.. </legal notes>

parameters
==========

*)

METHOD testBitXIsNotEqualTo
VAR_INPUT
	(* for the test it's the parameter ``currentValue`` *)
	valueToTest			:WORD;
	(* the bit number to check in this test, it's the parameter ``number``*)
	bitNumberToCheck	:CNM_AssertionInterfaces.BitNumberWord;
	(* this is the unexpected value of the bit ``bitNumberToCheck``, it's the parameter ``unexpectedValue`` *)
	bitIsSet			:BOOL;
END_VAR
VAR
	(* just the expectation if the assertion to test must be worng or true *)
	assertionIsWrong		:BOOL;
	(* bit with the number of ``bitNumberToCheck`` filtered from ``valueToTest`` *)
	specificBitOnly			:WORD;
	(* the bit number ``bitNumberToCheck`` is set to the value of ``bitIsSet`` only *)
	testBitOnly				:WORD;
	(* contains the format string for the test message *)
	message					:Tc2_System.T_MaxString;
	(* TwinCAT printf with the test message *)
	messageStringBuilder	:Tc2_Utilities.FB_FormatString;
END_VAR
THIS^.assertorContainer.resetAssertor();

specificBitOnly := (valueToTest AND SHL(THIS^.LSB_ONLY,bitNumberToCheck));
testBitOnly		:= SHL(TO_WORD(bitIsSet),bitNumberToCheck);
assertionIsWrong := (specificBitOnly = testBitOnly);

message := 'Bit number %d in currentValue: 16#%.4X ';
message := SEL(
	(specificBitOnly > THIS^.NO_BIT_SET),
	Tc2_Standard.CONCAT(message, 'is unset '),
	Tc2_Standard.CONCAT(message, 'is set ')
);
message := SEL(
	(testBitOnly > THIS^.NO_BIT_SET),
	Tc2_Standard.CONCAT(message, 'unexpectedValue: is unset (FALSE) '),
	Tc2_Standard.CONCAT(message, 'unexpectedValue: is set (TRUE)  ')
);
message := SEL(
	assertionIsWrong,
	Tc2_Standard.CONCAT(message, 'assertion must be TRUE'),
	Tc2_Standard.CONCAT(message, 'assertion must be FALSE')
);
messageStringBuilder(
	sFormat := message,
	arg1 := THIS^.AnyToArg(bitNumberToCheck),
	arg2 := THIS^.AnyToArg(valueToTest)
);

THIS^.assertorContainer.assertor.assert.bitNumber.simple.bitXIsNotEqualTo(
	currentValue 	:= valueToTest,
	number			:= bitNumberToCheck,
	unexpectedValue	:= bitIsSet,
	message			:= ''  
); 

THIS^.AssertEquals_BOOL(
	Expected 	:= assertionIsWrong,
	Actual 		:= THIS^.assertorContainer.wasAssertionWrong,
	Message 	:= messageStringBuilder.sOut
);
END_METHOD

(*

simple summary
==================
This test method tests ``assert.bitNumber.simple.bitXIsSet``
of CNM_AssertionInterfaces library, 
it provides the possibility to handover test data via parameter 


.. <legal notes>

legal notes
=================
| SPDX-FileCopyrightText: © 2022 ekvip automation GmbH <info@ekvip.de>
| SPDX-License-Identifier: Apache-2.0
| For details check: Apache-2.0_

.. _Apache-2.0: https://www.apache.org/licenses/LICENSE-2.0

.. </legal notes>

parameters
==========

*)

METHOD testBitXIsSet
VAR_INPUT
	(* for the test it's the parameter ``currentValue`` *)
	valueToTest			:WORD;
	(* the bit number to check in this test, it's the parameter ``number``*)
	bitNumberToCheck	:CNM_AssertionInterfaces.BitNumberWord;
END_VAR
VAR
	(* just the expectation if the assertion to test must be worng or true *)
	assertionIsWrong		:BOOL;
	(* contains the format string for the test message *)
	message					:Tc2_System.T_MaxString;
	(* TwinCAT printf with the test message *)
	messageStringBuilder	:Tc2_Utilities.FB_FormatString;
END_VAR
THIS^.assertorContainer.resetAssertor();

assertionIsWrong := ((valueToTest AND SHL(THIS^.LSB_ONLY,bitNumberToCheck)) = THIS^.NO_BIT_SET);

message := SEL(
	assertionIsWrong,
	'Bit number %d in currentValue: 16#%.4X is set assertion must be TRUE',
	'Bit number %d in currentValue: 16#%.4X is unset assertion must be FALSE'
);

messageStringBuilder(
	sFormat := message,
	arg1 := THIS^.AnyToArg(bitNumberToCheck),
	arg2 := THIS^.AnyToArg(valueToTest)
);

THIS^.assertorContainer.assertor.assert.bitNumber.simple.bitXIsSet(
	currentValue := valueToTest,
	number := bitNumberToCheck,
	message := ''
);

THIS^.AssertEquals_BOOL(
	Expected 	:= assertionIsWrong,
	Actual 		:= THIS^.assertorContainer.wasAssertionWrong,
	Message 	:= messageStringBuilder.sOut
);
END_METHOD

(*

simple summary
==================
This test method tests ``assert.bitNumber.simple.bitXIsUnset``
of CNM_AssertionInterfaces library, 
it provides the possibility to handover test data via parameter 


.. <legal notes>

legal notes
=================
| SPDX-FileCopyrightText: © 2022 ekvip automation GmbH <info@ekvip.de>
| SPDX-License-Identifier: Apache-2.0
| For details check: Apache-2.0_

.. _Apache-2.0: https://www.apache.org/licenses/LICENSE-2.0

.. </legal notes>

parameters
==========

*)

METHOD testBitXIsUnset
VAR_INPUT
	(* for the test it's the parameter ``currentValue`` *)
	valueToTest			:WORD;
	(* the bit number to check in this test, it's the parameter ``number``*)
	bitNumberToCheck	:CNM_AssertionInterfaces.BitNumberWord;
END_VAR
VAR
	(* just the expectation if the assertion to test must be worng or true *)
	assertionIsWrong		:BOOL;
	(* contains the format string for the test message *)
	message					:Tc2_System.T_MaxString;
	(* TwinCAT printf with the test message *)
	messageStringBuilder	:Tc2_Utilities.FB_FormatString;
END_VAR
THIS^.assertorContainer.resetAssertor();

assertionIsWrong := ((valueToTest AND SHL(THIS^.LSB_ONLY,bitNumberToCheck)) > THIS^.NO_BIT_SET);

message := SEL(
	assertionIsWrong,
	'Bit number %d in currentValue: 16#%.4X is unset assertion must be TRUE',
	'Bit number %d in currentValue: 16#%.4X is set assertion must be FALSE'
);

messageStringBuilder(
	sFormat := message,
	arg1 := THIS^.AnyToArg(bitNumberToCheck),
	arg2 := THIS^.AnyToArg(valueToTest)
);

THIS^.assertorContainer.assertor.assert.bitNumber.simple.bitXIsUnset(
	currentValue := valueToTest,
	number := bitNumberToCheck,
	message := ''
);

THIS^.AssertEquals_BOOL(
	Expected 	:= assertionIsWrong,
	Actual 		:= THIS^.assertorContainer.wasAssertionWrong,
	Message 	:= messageStringBuilder.sOut
);
END_METHOD

(*

simple summary
==================
This test method tests ``assert.bitNumber.simple.lsbIsEqualTo``
method of CNM_AssertionInterfaces library, 
it provides the possibility to handover test data via parameter 


.. <legal notes>

legal notes
=================
| SPDX-FileCopyrightText: © 2022 ekvip automation GmbH <info@ekvip.de>
| SPDX-License-Identifier: Apache-2.0
| For details check: Apache-2.0_

.. _Apache-2.0: https://www.apache.org/licenses/LICENSE-2.0

.. </legal notes>

parameters
==========

*)

METHOD testLsbIsEqualTo
VAR_INPUT
	(* for the test it's the parameter ``currentValue`` *)
	valueToTest		:WORD;
	(* for the test it's the parameter ``expectedValue`` *)
	expectedValue	:BOOL;
END_VAR
VAR
	(* just the expectation if the assertion to test must be worng or true *)
	assertionIsWrong		:BOOL;
	(* contains the format string for the test message *)
	message					:Tc2_System.T_MaxString;
	(* TwinCAT printf with the test message *)
	messageStringBuilder	:Tc2_Utilities.FB_FormatString;
END_VAR
THIS^.assertorContainer.resetAssertor();

assertionIsWrong := (valueToTest.FIRST_BIT <> expectedValue);
message := SEL(
	expectedValue,
	'currentValue: %d expectedValue is an unset (FALSE) assertion must be ',
	'currentValue: %d expectedValue is a set (TRUE) assertion must be '
);
message := SEL(
	assertionIsWrong,
	Tc2_Standard.CONCAT(message, 'TRUE'),
	Tc2_Standard.CONCAT(message, 'FALSE')
);

messageStringBuilder(
	sFormat := message,
	arg1 := THIS^.AnyToArg(valueToTest)
);

THIS^.assertorContainer.assertor.assert.bitNumber.simple.lsbIsEqualTo(
	currentValue 	:= valueToTest,
	expectedValue	:= expectedValue,
	message			:= ''  
); 

THIS^.AssertEquals_BOOL(
	Expected 	:= assertionIsWrong,
	Actual 		:= THIS^.assertorContainer.wasAssertionWrong,
	Message 	:= messageStringBuilder.sOut
);
END_METHOD

(*

simple summary
==================
This test method tests ``assert.bitNumber.simple.lsbIsNotEqualTo``
method of CNM_AssertionInterfaces library, 
it provides the possibility to handover test data via parameter 


.. <legal notes>

legal notes
=================
| SPDX-FileCopyrightText: © 2022 ekvip automation GmbH <info@ekvip.de>
| SPDX-License-Identifier: Apache-2.0
| For details check: Apache-2.0_

.. _Apache-2.0: https://www.apache.org/licenses/LICENSE-2.0

.. </legal notes>

parameters
==========

*)

METHOD testLsbIsNotEqualTo
VAR_INPUT
	(* for the test it's the parameter ``currentValue`` *)
	valueToTest	:WORD;
	(* for the test it's the parameter ``unexpectedValue`` *)
	unexpectedValue :BOOL;
END_VAR
VAR
	(* just the expectation if the assertion to test must be worng or true *)
	assertionIsWrong		:BOOL;
	(* contains the format string for the test message *)
	message					:Tc2_System.T_MaxString;
	(* TwinCAT printf with the test message *)
	messageStringBuilder	:Tc2_Utilities.FB_FormatString;
END_VAR
THIS^.assertorContainer.resetAssertor();

assertionIsWrong := (valueToTest.FIRST_BIT = unexpectedValue);
message := SEL(
	unexpectedValue,
	'currentValue: %d unexpectedValue is an unset (FALSE), assertion must be ',
	'currentValue: %d unexpectedValue is a set (TRUE) assertion must be '
);
message := SEL(
	assertionIsWrong,
	Tc2_Standard.CONCAT(message, 'TRUE'),
	Tc2_Standard.CONCAT(message, 'FALSE')
);

messageStringBuilder(
	sFormat := message,
	arg1 := THIS^.AnyToArg(valueToTest)
);

THIS^.assertorContainer.assertor.assert.bitNumber.simple.lsbIsNotEqualTo(
	currentValue 	:= valueToTest,
	unexpectedValue	:= unexpectedValue,
	message			:= ''  
); 

THIS^.AssertEquals_BOOL(
	Expected 	:= assertionIsWrong,
	Actual 		:= THIS^.assertorContainer.wasAssertionWrong,
	Message 	:= messageStringBuilder.sOut
);
END_METHOD

(*

simple summary
==================
This test method tests ``assert.bitNumber.simple.lsbIsSet``
of CNM_AssertionInterfaces library, 
it provides the possibility to handover test data via parameter 


.. <legal notes>

legal notes
=================
| SPDX-FileCopyrightText: © 2022 ekvip automation GmbH <info@ekvip.de>
| SPDX-License-Identifier: Apache-2.0
| For details check: Apache-2.0_

.. _Apache-2.0: https://www.apache.org/licenses/LICENSE-2.0

.. </legal notes>

parameters
==========

*)

METHOD testLsbIsSet
VAR_INPUT
	(* for the test it's the parameter ``currentValue`` *)
	valueToTest	:WORD;
END_VAR
VAR
	(* just the expectation if the assertion to test must be worng or true *)
	assertionIsWrong		:BOOL;
	(* contains the format string for the test message *)
	message					:Tc2_System.T_MaxString;
	(* TwinCAT printf with the test message *)
	messageStringBuilder	:Tc2_Utilities.FB_FormatString;
END_VAR
THIS^.assertorContainer.resetAssertor();

assertionIsWrong := (NOT valueToTest.FIRST_BIT);

message := SEL(
	assertionIsWrong,
	'currentValue is %d assertion must be TRUE',
	'currentValue is %d assertion must be FALSE'
);

messageStringBuilder(
	sFormat := message,
	arg1 := THIS^.AnyToArg(valueToTest)
);

THIS^.assertorContainer.assertor.assert.bitNumber.simple.lsbIsSet(
	currentValue 	:= valueToTest,
	message			:= ''  
); 

THIS^.AssertEquals_BOOL(
	Expected 	:= assertionIsWrong,
	Actual 		:= THIS^.assertorContainer.wasAssertionWrong,
	Message 	:= messageStringBuilder.sOut
);
END_METHOD

(*

simple summary
==================
This test method tests ``assert.bitNumber.simple.lsbIsUnset``
and ``assert.bitNumber.simple.lsbIsUnset``
of CNM_AssertionInterfaces library, 
it provides the possibility to handover test data via parameter 


.. <legal notes>

legal notes
=================
| SPDX-FileCopyrightText: © 2022 ekvip automation GmbH <info@ekvip.de>
| SPDX-License-Identifier: Apache-2.0
| For details check: Apache-2.0_

.. _Apache-2.0: https://www.apache.org/licenses/LICENSE-2.0

.. </legal notes>

parameters
==========

*)

METHOD testLsbIsUnset
VAR_INPUT
	(* for the test it's the parameter ``currentValue`` *)
	valueToTest	:WORD;
END_VAR
VAR
	(* just the expectation if the assertion to test must be worng or true *)
	assertionIsWrong		:BOOL;
	(* contains the format string for the test message *)
	message					:Tc2_System.T_MaxString;
	(* TwinCAT printf with the test message *)
	messageStringBuilder	:Tc2_Utilities.FB_FormatString;
END_VAR
THIS^.assertorContainer.resetAssertor();

assertionIsWrong := (valueToTest.FIRST_BIT);

message := SEL(
	assertionIsWrong,
	'currentValue is %d assertion must be TRUE',
	'currentValue is %d assertion must be FALSE'
);

messageStringBuilder(
	sFormat := message,
	arg1 := THIS^.AnyToArg(valueToTest)
);

THIS^.assertorContainer.assertor.assert.bitNumber.simple.lsbIsUnset(
	currentValue 	:= valueToTest,
	message			:= ''  
); 

THIS^.AssertEquals_BOOL(
	Expected 	:= assertionIsWrong,
	Actual 		:= THIS^.assertorContainer.wasAssertionWrong,
	Message 	:= messageStringBuilder.sOut
);
END_METHOD

(*

simple summary
==================
This test method tests ``assert.bitNumber.simple.msbIsEqualTo``
method of CNM_AssertionInterfaces library, 
it provides the possibility to handover test data via parameter 


.. <legal notes>

legal notes
=================
| SPDX-FileCopyrightText: © 2022 ekvip automation GmbH <info@ekvip.de>
| SPDX-License-Identifier: Apache-2.0
| For details check: Apache-2.0_

.. _Apache-2.0: https://www.apache.org/licenses/LICENSE-2.0

.. </legal notes>

parameters
==========

*)

METHOD testMsbIsEqualTo
VAR_INPUT
	(* for the test it's the parameter ``currentValue`` *)
	valueToTest		:WORD;
	(* for the test it's the parameter ``expectedValue`` *)
	expectedValue	:BOOL;
END_VAR
VAR
	(* just the expectation if the assertion to test must be worng or true *)
	assertionIsWrong		:BOOL;
	(* contains the format string for the test message *)
	message					:Tc2_System.T_MaxString;
	(* TwinCAT printf with the test message *)
	messageStringBuilder	:Tc2_Utilities.FB_FormatString;
END_VAR
THIS^.assertorContainer.resetAssertor();

assertionIsWrong := (valueToTest.LAST_BIT <> expectedValue);

message := SEL(
	expectedValue,
	'currentValue: 16#%.4X expectedValue is an unset (FALSE) assertion must be ',
	'currentValue: 16#%.4X expectedValue is a set (TRUE) assertion must be '
);
message := SEL(
	assertionIsWrong,
	Tc2_Standard.CONCAT(message, 'TRUE'),
	Tc2_Standard.CONCAT(message, 'FALSE')
);

messageStringBuilder(
	sFormat := message,
	arg1 := THIS^.AnyToArg(valueToTest)
);

THIS^.assertorContainer.assertor.assert.bitNumber.simple.msbIsEqualTo(
	currentValue 	:= valueToTest,
	expectedValue	:= expectedValue,
	message			:= ''  
); 

THIS^.AssertEquals_BOOL(
	Expected 	:= assertionIsWrong,
	Actual 		:= THIS^.assertorContainer.wasAssertionWrong,
	Message 	:= messageStringBuilder.sOut
);
END_METHOD

(*

simple summary
==================
This test method tests ``assert.bitNumber.simple.msbIsNotEqualTo``
method of CNM_AssertionInterfaces library, 
it provides the possibility to handover test data via parameter 


.. <legal notes>

legal notes
=================
| SPDX-FileCopyrightText: © 2022 ekvip automation GmbH <info@ekvip.de>
| SPDX-License-Identifier: Apache-2.0
| For details check: Apache-2.0_

.. _Apache-2.0: https://www.apache.org/licenses/LICENSE-2.0

.. </legal notes>

parameters
==========

*)

METHOD testMsbIsNotEqualTo
VAR_INPUT
	(* for the test it's the parameter ``currentValue`` *)
	valueToTest	:WORD;
	(* for the test it's the parameter ``unexpectedValue`` *)
	unexpectedValue :BOOL;
END_VAR
VAR
	(* just the expectation if the assertion to test must be worng or true *)
	assertionIsWrong		:BOOL;
	(* contains the format string for the test message *)
	message					:Tc2_System.T_MaxString;
	(* TwinCAT printf with the test message *)
	messageStringBuilder	:Tc2_Utilities.FB_FormatString;
END_VAR
THIS^.assertorContainer.resetAssertor();

assertionIsWrong := (valueToTest.LAST_BIT = unexpectedValue);

message := SEL(
	unexpectedValue,
	'currentValue: 16#%.4X unexpectedValue is an unset (FALSE) assertion must be ',
	'currentValue: 16#%.4X unexpectedValue is a set (TRUE) assertion must be '
);
message := SEL(
	assertionIsWrong,
	Tc2_Standard.CONCAT(message, 'TRUE'),
	Tc2_Standard.CONCAT(message, 'FALSE')
);

messageStringBuilder(
	sFormat := message,
	arg1 := THIS^.AnyToArg(valueToTest)
);

THIS^.assertorContainer.assertor.assert.bitNumber.simple.msbIsNotEqualTo(
	currentValue 	:= valueToTest,
	unexpectedValue	:= unexpectedValue,
	message			:= ''  
); 

THIS^.AssertEquals_BOOL(
	Expected 	:= assertionIsWrong,
	Actual 		:= THIS^.assertorContainer.wasAssertionWrong,
	Message 	:= messageStringBuilder.sOut
);
END_METHOD

(*

simple summary
==================
This test method tests ``assert.bitNumber.simple.msbIsSet``
of CNM_AssertionInterfaces library, 
it provides the possibility to handover test data via parameter 


.. <legal notes>

legal notes
=================
| SPDX-FileCopyrightText: © 2022 ekvip automation GmbH <info@ekvip.de>
| SPDX-License-Identifier: Apache-2.0
| For details check: Apache-2.0_

.. _Apache-2.0: https://www.apache.org/licenses/LICENSE-2.0

.. </legal notes>

parameters
==========

*)

METHOD testMsbIsSet
VAR_INPUT
	(* for the test it's the parameter ``currentValue`` *)
	valueToTest	:WORD;
END_VAR
VAR
	(* just the expectation if the assertion to test must be worng or true *)
	assertionIsWrong		:BOOL;
	(* contains the format string for the test message *)
	message					:Tc2_System.T_MaxString;
	(* TwinCAT printf with the test message *)
	messageStringBuilder	:Tc2_Utilities.FB_FormatString;
END_VAR
THIS^.assertorContainer.resetAssertor();

assertionIsWrong := (NOT valueToTest.LAST_BIT);

message := SEL(
	assertionIsWrong,
	'currentValue is 16#%.4X assertion must be TRUE',
	'currentValue is 16#%.4X assertion must be FALSE'
);

messageStringBuilder(
	sFormat := message,
	arg1 := THIS^.AnyToArg(valueToTest)
);

THIS^.assertorContainer.assertor.assert.bitNumber.simple.msbIsSet(
	currentValue 	:= valueToTest,
	message			:= ''  
); 

THIS^.AssertEquals_BOOL(
	Expected 	:= assertionIsWrong,
	Actual 		:= THIS^.assertorContainer.wasAssertionWrong,
	Message 	:= messageStringBuilder.sOut
);
END_METHOD

(*

simple summary
==================
This test method tests ``assert.bitNumber.simple.msbIsUnset``
of CNM_AssertionInterfaces library, 
it provides the possibility to handover test data via parameter 


.. <legal notes>

legal notes
=================
| SPDX-FileCopyrightText: © 2022 ekvip automation GmbH <info@ekvip.de>
| SPDX-License-Identifier: Apache-2.0
| For details check: Apache-2.0_

.. _Apache-2.0: https://www.apache.org/licenses/LICENSE-2.0

.. </legal notes>

parameters
==========

*)

METHOD testMsbIsUnset
VAR_INPUT
	(* for the test it's the parameter ``currentValue`` *)
	valueToTest	:WORD;
END_VAR
VAR
	(* just the expectation if the assertion to test must be worng or true *)
	assertionIsWrong		:BOOL;
	(* contains the format string for the test message *)
	message					:Tc2_System.T_MaxString;
	(* TwinCAT printf with the test message *)
	messageStringBuilder	:Tc2_Utilities.FB_FormatString;
END_VAR
THIS^.assertorContainer.resetAssertor();

assertionIsWrong := (valueToTest.LAST_BIT);

message := SEL(
	assertionIsWrong,
	'currentValue is 16#%.4X assertion must be TRUE',
	'currentValue is 16#%.4X assertion must be FALSE'
);

messageStringBuilder(
	sFormat := message,
	arg1 := THIS^.AnyToArg(valueToTest)
);

THIS^.assertorContainer.assertor.assert.bitNumber.simple.msbIsUnset(
	currentValue 	:= valueToTest,
	message			:= ''  
); 

THIS^.AssertEquals_BOOL(
	Expected 	:= assertionIsWrong,
	Actual 		:= THIS^.assertorContainer.wasAssertionWrong,
	Message 	:= messageStringBuilder.sOut
);
END_METHOD

(*

simple summary
==================
This test method tests ``assert.bitNumber.simple.orMaskIsEqualTo``
method of CNM_AssertionInterfaces library, 
it provides the possibility to handover test data via parameter 


.. <legal notes>

legal notes
=================
| SPDX-FileCopyrightText: © 2022 ekvip automation GmbH <info@ekvip.de>
| SPDX-License-Identifier: Apache-2.0
| For details check: Apache-2.0_

.. _Apache-2.0: https://www.apache.org/licenses/LICENSE-2.0

.. </legal notes>

parameters
==========

*)

METHOD testOrMaskIsEqualTo 
VAR_INPUT
	(* for the test it's the parameter ``currentValue`` *)
	valueToTest	:WORD;
	(* it's the mask for the currentValue *)
	mask		:WORD;
	(* for the test it's the parameter ``expectedValue`` *)
	expected	:WORD;
END_VAR
VAR
	(* just the expectation if the assertion to test must be worng or true *)
	assertionIsWrong		:BOOL;
	(* result of the bit operation to determine the value of ``assertionIsWrong`` *)
	result					:WORD;
	(* contains the format string for the test message *)
	message					:Tc2_System.T_MaxString;
	(* TwinCAT printf with the test message *)
	messageStringBuilder	:Tc2_Utilities.FB_FormatString;
END_VAR
THIS^.assertorContainer.resetAssertor();

result := (valueToTest OR mask);
assertionIsWrong := (result <> expected);
message := SEL(
	assertionIsWrong,
	'currentValue: 16#%.4X OR mask: 16#%.4X is 16#%.4X expectedValue: 16#%.4X assertion must be TRUE', 
	'currentValue: 16#%.4X OR mask: 16#%.4X is 16#%.4X expectedValue: 16#%.4X assertion must be FALSE'
);
messageStringBuilder(
	sFormat := message,
	arg1 := THIS^.AnyToArg(valueToTest),
	arg2 := THIS^.AnyToArg(mask),
	arg3 := THIS^.AnyToArg(result),
	arg4 := THIS^.AnyToArg(expected)
);

THIS^.assertorContainer.assertor.assert.bitNumber.simple.orMaskIsEqualTo(
	currentValue	:= valueToTest,
	mask 			:= mask,
	expectedValue	:= expected,
	message			:= ''
);

THIS^.AssertEquals_BOOL(
	Expected 	:= assertionIsWrong,
	Actual 		:= THIS^.assertorContainer.wasAssertionWrong,
	Message 	:= messageStringBuilder.sOut
);
END_METHOD

(*

simple summary
==================
This test method tests ``assert.bitNumber.simple.orMaskIsNotEqualTo``
method of CNM_AssertionInterfaces library, 
it provides the possibility to handover test data via parameter 


.. <legal notes>

legal notes
=================
| SPDX-FileCopyrightText: © 2022 ekvip automation GmbH <info@ekvip.de>
| SPDX-License-Identifier: Apache-2.0
| For details check: Apache-2.0_

.. _Apache-2.0: https://www.apache.org/licenses/LICENSE-2.0

.. </legal notes>

parameters
==========

*)

METHOD testOrMaskIsNotEqualTo 
VAR_INPUT
	(* for the test it's the parameter ``currentValue`` *)
	valueToTest	:WORD;
	(* it's the mask for the currentValue *)
	mask		:WORD;
	(* for the test it's the parameter ``unexpectedValue`` *)
	unexpected	:WORD;
END_VAR
VAR
	(* just the expectation if the assertion to test must be worng or true *)
	assertionIsWrong		:BOOL;
	(* result of the bit operation to determine the value of ``assertionIsWrong`` *)
	result					:WORD;
	(* contains the format string for the test message *)
	message					:Tc2_System.T_MaxString;
	(* TwinCAT printf with the test message *)
	messageStringBuilder	:Tc2_Utilities.FB_FormatString;
END_VAR
THIS^.assertorContainer.resetAssertor();

result := (valueToTest OR mask);
assertionIsWrong := (result = unexpected);
message := SEL(
	assertionIsWrong,
	'currentValue: 16#%.4X OR mask: 16#%.4X is 16#%.4X unexpectedValue: 16#%.4X assertion must be TRUE', 
	'currentValue: 16#%.4X OR mask: 16#%.4X is 16#%.4X unexpectedValue: 16#%.4X assertion must be FALSE'
);
messageStringBuilder(
	sFormat := message,
	arg1 := THIS^.AnyToArg(valueToTest),
	arg2 := THIS^.AnyToArg(mask),
	arg3 := THIS^.AnyToArg(result),
	arg4 := THIS^.AnyToArg(unexpected)
);

THIS^.assertorContainer.assertor.assert.bitNumber.simple.orMaskIsNotEqualTo(
	currentValue	:= valueToTest,
	mask 			:= mask,
	unexpectedValue	:= unexpected,
	message			:= ''
);

THIS^.AssertEquals_BOOL(
	Expected 	:= assertionIsWrong,
	Actual 		:= THIS^.assertorContainer.wasAssertionWrong,
	Message 	:= messageStringBuilder.sOut
);
END_METHOD

(*

simple summary
==================
This test method tests ``assert.bitNumber.simple.valueIsEqualTo``
method of CNM_AssertionInterfaces library, 
it provides the possibility to handover test data via parameter 


.. <legal notes>

legal notes
=================
| SPDX-FileCopyrightText: © 2022 ekvip automation GmbH <info@ekvip.de>
| SPDX-License-Identifier: Apache-2.0
| For details check: Apache-2.0_

.. _Apache-2.0: https://www.apache.org/licenses/LICENSE-2.0

.. </legal notes>

parameters
==========

*)

METHOD testValueIsEqualTo
VAR_INPUT
	(* for the test it's the parameter ``currentValue`` *)
	valueToTest	:WORD;
	(* for the test it's the parameter ``expectedValue`` *)
	expected	:WORD;
END_VAR
VAR
	(* just the expectation if the assertion to test must be worng or true *)
	assertionIsWrong		:BOOL;
	(* contains the format string for the test message *)
	message					:Tc2_System.T_MaxString;
	(* TwinCAT printf with the test message *)
	messageStringBuilder	:Tc2_Utilities.FB_FormatString;
END_VAR
THIS^.assertorContainer.resetAssertor();

assertionIsWrong := (valueToTest <> expected);
message := SEL(
	assertionIsWrong,
	'currentValue is %d expectedValue is %d assertion must be TRUE', 
	'currentValue is %d expectedValue is %d assertion must be FALSE'
);
messageStringBuilder(
	sFormat := message,
	arg1 := THIS^.AnyToArg(valueToTest),
	arg2 := THIS^.AnyToArg(expected)
);

THIS^.assertorContainer.assertor.assert.bitNumber.simple.valueIsEqualTo(
	currentValue := valueToTest,
	expectedValue := expected,
	message := ''
);

THIS^.AssertEquals_BOOL(
	Expected 	:= assertionIsWrong,
	Actual 		:= THIS^.assertorContainer.wasAssertionWrong,
	Message 	:= messageStringBuilder.sOut
);
END_METHOD

(*

simple summary
==================
This test method tests ``assert.bitNumber.simple.valueIsGreaterThan``
method of CNM_AssertionInterfaces library, 
it provides the possibility to handover test data via parameter 


.. <legal notes>

legal notes
=================
| SPDX-FileCopyrightText: © 2022 ekvip automation GmbH <info@ekvip.de>
| SPDX-License-Identifier: Apache-2.0
| For details check: Apache-2.0_

.. _Apache-2.0: https://www.apache.org/licenses/LICENSE-2.0

.. </legal notes>

parameters
==========

*)

METHOD testValueIsGreater
VAR_INPUT
	(* for the test it's the parameter ``currentValue`` *)
	valueToTest	:WORD;
	(* for the test it's the parameter ``lessValue`` *)
	less		:WORD;
END_VAR
VAR
	(* just the expectation if the assertion to test must be worng or true *)
	assertionIsWrong		:BOOL;
	(* contains the format string for the test message *)
	message					:Tc2_System.T_MaxString;
	(* TwinCAT printf with the test message *)
	messageStringBuilder	:Tc2_Utilities.FB_FormatString;
END_VAR
THIS^.assertorContainer.resetAssertor();

assertionIsWrong := (valueToTest <= less);
message := SEL(
	assertionIsWrong,
	'currentValue is %d lessValue is %d assertion must be TRUE', 
	'currentValue is %d lessValue is %d assertion must be FALSE'
);
messageStringBuilder(
	sFormat := message,
	arg1 := THIS^.AnyToArg(valueToTest),
	arg2 := THIS^.AnyToArg(less)
);

THIS^.assertorContainer.assertor.assert.bitNumber.simple.valueIsGreaterThan(
	currentValue := valueToTest,
	lessValue := less,
	message := ''
);

THIS^.AssertEquals_BOOL(
	Expected 	:= assertionIsWrong,
	Actual 		:= THIS^.assertorContainer.wasAssertionWrong,
	Message 	:= messageStringBuilder.sOut
);
END_METHOD

(*

simple summary
==================
This test method tests ``assert.bitNumber.simple.valueIsInRangeOf``
method of CNM_AssertionInterfaces library, 
it provides the possibility to handover test data via parameter 


.. <legal notes>

legal notes
=================
| SPDX-FileCopyrightText: © 2022 ekvip automation GmbH <info@ekvip.de>
| SPDX-License-Identifier: Apache-2.0
| For details check: Apache-2.0_

.. _Apache-2.0: https://www.apache.org/licenses/LICENSE-2.0

.. </legal notes>

parameters
==========

*)

METHOD testValueIsInRangeOf
VAR_INPUT
	(* for the test it's the parameter ``lowerLimit`` *)
	lower		:WORD;
	(* for the test it's the parameter ``currentValue`` *)
	valueToTest	:WORD;
	(* for the test it's the parameter ``upperLimit`` *)
	upper		:WORD;
END_VAR          
VAR
	(* just the expectation if the assertion to test must be worng or true *)
	assertionIsWrong		:BOOL;
	(* contains the format string for the test message *)
	message					:Tc2_System.T_MaxString;
	(* TwinCAT printf with the test message *)
	messageStringBuilder	:Tc2_Utilities.FB_FormatString;
END_VAR
THIS^.assertorContainer.resetAssertor();

assertionIsWrong := ((valueToTest < lower) OR (valueToTest > upper)); 

message := SEL(
	assertionIsWrong,
	'lowerLimit is %d currentValue is %d upperLimit is %d assertion must be TRUE', 
	'lowerLimit is %d currentValue is %d upperLimit is %d assertion must be FALSE'
);

messageStringBuilder(
	sFormat := message,
	arg1 := THIS^.AnyToArg(lower),
	arg2 := THIS^.AnyToArg(valueToTest),
	arg3 := THIS^.AnyToArg(upper)
);

THIS^.assertorContainer.assertor.assert.bitNumber.simple.valueIsInRangeOf(
	lowerLimit := lower,
	currentValue := valueToTest,
	upperLimit := upper,
	message := ''
);

THIS^.AssertEquals_BOOL(
	Expected 	:= assertionIsWrong,
	Actual 		:= THIS^.assertorContainer.wasAssertionWrong,
	Message 	:= messageStringBuilder.sOut
);
END_METHOD

(*

simple summary
==================
This test method tests ``assert.bitNumber.simple.valueIsLessThan``
method of CNM_AssertionInterfaces library, 
it provides the possibility to handover test data via parameter 


.. <legal notes>

legal notes
=================
| SPDX-FileCopyrightText: © 2022 ekvip automation GmbH <info@ekvip.de>
| SPDX-License-Identifier: Apache-2.0
| For details check: Apache-2.0_

.. _Apache-2.0: https://www.apache.org/licenses/LICENSE-2.0

.. </legal notes>

parameters
==========

*)

METHOD testValueIsLessThan
VAR_INPUT
	(* for the test it's the parameter ``currentValue`` *)
	valueToTest	:WORD;
	(* for the test it's the parameter ``greaterValue`` *)
	greater		:WORD;
END_VAR
VAR
	(* just the expectation if the assertion to test must be worng or true *)
	assertionIsWrong		:BOOL;
	(* contains the format string for the test message *)
	message					:Tc2_System.T_MaxString;
	(* TwinCAT printf with the test message *)
	messageStringBuilder	:Tc2_Utilities.FB_FormatString;
END_VAR
THIS^.assertorContainer.resetAssertor();

assertionIsWrong := (valueToTest >= greater);
message := SEL(
	assertionIsWrong,
	'currentValue is %d greaterValue is %d assertion must be TRUE',
	'currentValue is %d greaterValue is %d assertion must be FALSE'
);
messageStringBuilder(
	sFormat := message,
	arg1 := THIS^.AnyToArg(valueToTest),
	arg2 := THIS^.AnyToArg(greater)
);

THIS^.assertorContainer.assertor.assert.bitNumber.simple.valueIsLessThan(
	currentValue := valueToTest,
	greaterValue := greater,
	message := ''
);

THIS^.AssertEquals_BOOL(
	Expected 	:= assertionIsWrong,
	Actual 		:= THIS^.assertorContainer.wasAssertionWrong,
	Message 	:= messageStringBuilder.sOut
);
END_METHOD

(*

simple summary
==================
This test method tests ``assert.bitNumber.simple.valueIsMax``
method of CNM_AssertionInterfaces library, 
it provides the possibility to handover test data via parameter 


.. <legal notes>

legal notes
=================
| SPDX-FileCopyrightText: © 2022 ekvip automation GmbH <info@ekvip.de>
| SPDX-License-Identifier: Apache-2.0
| For details check: Apache-2.0_

.. _Apache-2.0: https://www.apache.org/licenses/LICENSE-2.0

.. </legal notes>

parameters
==========

*)

METHOD testValueIsMax 
VAR_INPUT
	(* for the test it's the parameter ``currentValue`` *)
	valueToTest	:WORD;
	(* for the test it's the parameter ``maximumValue`` *)
	maximum		:WORD;
END_VAR
VAR
	(* just the expectation if the assertion to test must be worng or true *)
	assertionIsWrong		:BOOL;
	(* contains the format string for the test message *)
	message					:Tc2_System.T_MaxString;
	(* TwinCAT printf with the test message *)
	messageStringBuilder	:Tc2_Utilities.FB_FormatString;
END_VAR
THIS^.assertorContainer.resetAssertor();

assertionIsWrong := (valueToTest > maximum);
message := SEL(
	assertionIsWrong,
	'currentValue is %d maximumValue is %d assertion must be TRUE',
	'currentValue is %d maximumValue is %d assertion must be FALSE'
);
messageStringBuilder(
	sFormat := message,
	arg1 := THIS^.AnyToArg(valueToTest),
	arg2 := THIS^.AnyToArg(maximum)
);

THIS^.assertorContainer.assertor.assert.bitNumber.simple.valueIsMax(
	currentValue := valueToTest,
	maximumValue := maximum,
	message := ''
);

THIS^.AssertEquals_BOOL(
	Expected 	:= assertionIsWrong,
	Actual 		:= THIS^.assertorContainer.wasAssertionWrong,
	Message 	:= messageStringBuilder.sOut
);
END_METHOD

(*

simple summary
==================
This test method tests ``assert.bitNumber.simple.valueIsMin``
method of CNM_AssertionInterfaces library, 
it provides the possibility to handover test data via parameter 


.. <legal notes>

legal notes
=================
| SPDX-FileCopyrightText: © 2022 ekvip automation GmbH <info@ekvip.de>
| SPDX-License-Identifier: Apache-2.0
| For details check: Apache-2.0_

.. _Apache-2.0: https://www.apache.org/licenses/LICENSE-2.0

.. </legal notes>

parameters
==========

*)

METHOD testValueIsMin 
VAR_INPUT
	(* for the test it's the parameter ``currentValue`` *)
	valueToTest	:WORD;
	(* for the test it's the parameter ``minimumValue`` *)
	minimum		:WORD;
END_VAR
VAR
	(* just the expectation if the assertion to test must be worng or true *)
	assertionIsWrong		:BOOL;
	(* contains the format string for the test message *)
	message					:Tc2_System.T_MaxString;
	(* TwinCAT printf with the test message *)
	messageStringBuilder	:Tc2_Utilities.FB_FormatString;
END_VAR
THIS^.assertorContainer.resetAssertor();

assertionIsWrong := (valueToTest < minimum);
message := SEL(
	assertionIsWrong,
	'currentValue is %d minimumValue is %d assertion must be TRUE',
	'currentValue is %d minimumValue is %d assertion must be FALSE'
);
messageStringBuilder(
	sFormat := message,
	arg1 := THIS^.AnyToArg(valueToTest),
	arg2 := THIS^.AnyToArg(minimum)
);

THIS^.assertorContainer.assertor.assert.bitNumber.simple.valueIsMin(
	currentValue := valueToTest,
	minimumValue := minimum,
	message := ''
);

THIS^.AssertEquals_BOOL(
	Expected 	:= assertionIsWrong,
	Actual 		:= THIS^.assertorContainer.wasAssertionWrong,
	Message 	:= messageStringBuilder.sOut
);
END_METHOD

(*

simple summary
==================
This test method tests ``assert.bitNumber.simple.valueIsNotEqualTo``
method of CNM_AssertionInterfaces library, 
it provides the possibility to handover test data via parameter 


.. <legal notes>

legal notes
=================
| SPDX-FileCopyrightText: © 2022 ekvip automation GmbH <info@ekvip.de>
| SPDX-License-Identifier: Apache-2.0
| For details check: Apache-2.0_

.. _Apache-2.0: https://www.apache.org/licenses/LICENSE-2.0

.. </legal notes>

parameters
==========

*)

METHOD testValueIsNotEqualTo
VAR_INPUT
	(* for the test it's the parameter ``currentValue`` *)
	valueToTest	:WORD;
	(* for the test it's the parameter ``unexpectedValue`` *)
	unexpected	:WORD;
END_VAR
VAR
	(* just the expectation if the assertion to test must be worng or true *)
	assertionIsWrong		:BOOL;
	(* contains the format string for the test message *)
	message					:Tc2_System.T_MaxString;
	(* TwinCAT printf with the test message *)
	messageStringBuilder	:Tc2_Utilities.FB_FormatString;
END_VAR
THIS^.assertorContainer.resetAssertor();

assertionIsWrong := (valueToTest = unexpected);
message := SEL(
	assertionIsWrong,
	'currentValue is %d unexpectedValue is %d assertion must be TRUE', 
	'currentValue is %d unexpectedValue is %d assertion must be FALSE'
);
messageStringBuilder(
	sFormat := message,
	arg1 := THIS^.AnyToArg(valueToTest),
	arg2 := THIS^.AnyToArg(unexpected)
);

THIS^.assertorContainer.assertor.assert.bitNumber.simple.valueIsNotEqualTo(
	currentValue := valueToTest,
	unexpectedValue := unexpected,
	message := ''
);

THIS^.AssertEquals_BOOL(
	Expected 	:= assertionIsWrong,
	Actual 		:= THIS^.assertorContainer.wasAssertionWrong,
	Message 	:= messageStringBuilder.sOut
);
END_METHOD

(*

simple summary
==================
This test method tests ``assert.bitNumber.simple.xorMaskIsEqualTo``
method of CNM_AssertionInterfaces library, 
it provides the possibility to handover test data via parameter 


.. <legal notes>

legal notes
=================
| SPDX-FileCopyrightText: © 2022 ekvip automation GmbH <info@ekvip.de>
| SPDX-License-Identifier: Apache-2.0
| For details check: Apache-2.0_

.. _Apache-2.0: https://www.apache.org/licenses/LICENSE-2.0

.. </legal notes>

parameters
==========

*)

METHOD testXorMaskIsEqualTo 
VAR_INPUT
	(* for the test it's the parameter ``currentValue`` *)
	valueToTest	:WORD;
	(* it's the mask for the currentValue *)
	mask		:WORD;
	(* for the test it's the parameter ``expectedValue`` *)
	expected	:WORD;
END_VAR
VAR
	(* just the expectation if the assertion to test must be worng or true *)
	assertionIsWrong		:BOOL;
	(* result of the bit operation to determine the value of ``assertionIsWrong`` *)
	result					:WORD;
	(* contains the format string for the test message *)
	message					:Tc2_System.T_MaxString;
	(* TwinCAT printf with the test message *)
	messageStringBuilder	:Tc2_Utilities.FB_FormatString;
END_VAR
THIS^.assertorContainer.resetAssertor();

result := (valueToTest XOR mask);
assertionIsWrong := (result <> expected);
message := SEL(
	assertionIsWrong,
	'currentValue: 16#%.4X XOR mask: 16#%.4X is 16#%.4X expectedValue: 16#%.4X assertion must be TRUE', 
	'currentValue: 16#%.4X XOR mask: 16#%.4X is 16#%.4X expectedValue: 16#%.4X assertion must be FALSE'
);
messageStringBuilder(
	sFormat := message,
	arg1 := THIS^.AnyToArg(valueToTest),
	arg2 := THIS^.AnyToArg(mask),
	arg3 := THIS^.AnyToArg(result),
	arg4 := THIS^.AnyToArg(expected)
);

THIS^.assertorContainer.assertor.assert.bitNumber.simple.xorMaskIsEqualTo(
	currentValue	:= valueToTest,
	mask 			:= mask,
	expectedValue	:= expected,
	message			:= ''
);

THIS^.AssertEquals_BOOL(
	Expected 	:= assertionIsWrong,
	Actual 		:= THIS^.assertorContainer.wasAssertionWrong,
	Message 	:= messageStringBuilder.sOut
);
END_METHOD

(*

simple summary
==================
This test method tests ``assert.bitNumber.simple.xorMaskIsNotEqualTo``
method of CNM_AssertionInterfaces library, 
it provides the possibility to handover test data via parameter 


.. <legal notes>

legal notes
=================
| SPDX-FileCopyrightText: © 2022 ekvip automation GmbH <info@ekvip.de>
| SPDX-License-Identifier: Apache-2.0
| For details check: Apache-2.0_

.. _Apache-2.0: https://www.apache.org/licenses/LICENSE-2.0

.. </legal notes>

parameters
==========

*)

METHOD testXorMaskIsNotEqualTo 
VAR_INPUT
	(* for the test it's the parameter ``currentValue`` *)
	valueToTest	:WORD;
	(* it's the mask for the currentValue *)
	mask		:WORD;
	(* for the test it's the parameter ``unexpectedValue`` *)
	unexpected	:WORD;
END_VAR
VAR
	(* just the expectation if the assertion to test must be worng or true *)
	assertionIsWrong		:BOOL;
	(* result of the bit operation to determine the value of ``assertionIsWrong`` *)
	result					:WORD;
	(* contains the format string for the test message *)
	message					:Tc2_System.T_MaxString;
	(* TwinCAT printf with the test message *)
	messageStringBuilder	:Tc2_Utilities.FB_FormatString;
END_VAR
THIS^.assertorContainer.resetAssertor();

result := (valueToTest XOR mask);
assertionIsWrong := (result = unexpected);
message := SEL(
	assertionIsWrong,
	'currentValue: 16#%.4X XOR mask: 16#%.4X is 16#%.4X unexpectedValue: 16#%.4X assertion must be TRUE', 
	'currentValue: 16#%.4X XOR mask: 16#%.4X is 16#%.4X unexpectedValue: 16#%.4X assertion must be FALSE'
);
messageStringBuilder(
	sFormat := message,
	arg1 := THIS^.AnyToArg(valueToTest),
	arg2 := THIS^.AnyToArg(mask),
	arg3 := THIS^.AnyToArg(result),
	arg4 := THIS^.AnyToArg(unexpected)
);

THIS^.assertorContainer.assertor.assert.bitNumber.simple.xorMaskIsNotEqualTo(
	currentValue	:= valueToTest,
	mask 			:= mask,
	unexpectedValue	:= unexpected,
	message			:= ''
);

THIS^.AssertEquals_BOOL(
	Expected 	:= assertionIsWrong,
	Actual 		:= THIS^.assertorContainer.wasAssertionWrong,
	Message 	:= messageStringBuilder.sOut
);
END_METHOD

END_FUNCTION_BLOCK

// ---- AssertionTester/AssertionTests/DateTimeAssertions/classes/DTAssertionTests.TcPOU
(*

short summary
==================
This class tests all methods of DT assertions
with various combinations of inputs and checks expected 
outputs are satisfied or not

.. <legal notes>

legal notes
=================
| SPDX-FileCopyrightText: © 2022 ekvip automation GmbH <info@ekvip.de>
| SPDX-License-Identifier: Apache-2.0
| For details check: Apache-2.0_

.. _Apache-2.0: https://www.apache.org/licenses/LICENSE-2.0

.. </legal notes>

methods and properties
======================

*)


FUNCTION_BLOCK DTAssertionTests EXTENDS AbstractAssertorTest
VAR
	
END_VAR
VAR CONSTANT
	(* prefix to unify the test names *)
	TEST_NAME_PREFIX		:STRING := 'assert.dateAndTime.simple.dateAndTime.';
	(* max value of a DWORD *)
	{attribute 'hide'}
	MAX_DWORD				:DWORD := 16#FFFF_FFFF;
	(* min value of a DWORD *)
	{attribute 'hide'}
	MIN_DWORD				:DWORD := 16#0000_0000;
	(* only the msb is set *)
	{attribute 'hide'}
	MSB_ONLY				:DWORD := 16#8000_0000;
	(* only the msb is set *)
	{attribute 'hide'}
	LSB_ONLY				:DWORD := 16#0000_0001;
	(* all bits set except the msb *)
	{attribute 'hide'}
	WITHOUT_MSB 			:DWORD := 16#7FFF_FFFF;
	(* for every nibble is the msb set only *)
	{attribute 'hide'}
	ALL_NIBBLE_MSB			:DWORD := 16#8888_8888;
	(* for every nibble is the msb unset only *)
	{attribute 'hide'}
	WITHOUT_NIBBLE_MSB		:DWORD := 16#7777_7777;
	(* for every nibble is the lsb set only *)
	{attribute 'hide'}
	ALL_NIBBLE_LSB			:DWORD := 16#1111_1111;
	(* every bit is set except the lsb *)
	{attribute 'hide'}
	LSB_IS_UNSET			:DWORD := 16#FFFF_FFFE;
	(* max vale of date and time *)
	DT_MAX					:DT := TO_DT(MAX_DWORD);
	(* min vale of date and time *)
	DT_MIN					:DT := TO_DT(MIN_DWORD);
	(* only the msb is set *)
	DT_MSB_ONLY				:DT := TO_DT(MSB_ONLY);
	(* all bits set except the msb *)
	DT_WITHOUT_MSB 			:DT := TO_DT(WITHOUT_MSB);
	(* for every nibble is the msb set only *)
	DT_ALL_NIBBLE_MSB		:DT := TO_DT(ALL_NIBBLE_MSB);
	(* for every nibble is the msb unset only *)
	DT_WITHOUT_NIBBLE_MSB	:DT := TO_DT(WITHOUT_NIBBLE_MSB);
	(* for every nibble is the lsb set only *)
	DT_ALL_NIBBLE_LSB		:DT := TO_DT(ALL_NIBBLE_LSB);	
	(* every bit is set except the lsb *)
	DT_LSB_IS_UNSET			:DT := TO_DT(LSB_IS_UNSET);
	(* only the msb is set *)
	DT_LSB_ONLY				:DT := TO_DT(LSB_ONLY);
END_VAR

THIS^.runValueIsEqualToTests();
THIS^.runValueIsGreaterThanTests();
THIS^.runValueIsInRangeOfTests();
THIS^.runValueIsLessThanTests();
THIS^.runValueIsMaxTests();
THIS^.runValueIsMinTests();
THIS^.runValueIsNotEqualToTests();

(*

short summary
==================
This test method is a helper function to create a unified test name

.. <legal notes>

legal notes
=================
| SPDX-FileCopyrightText: © 2022 ekvip automation GmbH <info@ekvip.de>
| SPDX-License-Identifier: Apache-2.0
| For details check: Apache-2.0_

.. _Apache-2.0: https://www.apache.org/licenses/LICENSE-2.0

.. </legal notes>

parameters
==========

*)

METHOD PROTECTED getTestNameFor :Tc2_System.T_MaxString
VAR_INPUT
	(* name of the method to test, to create a unified test name *)
	nameOfMethodToTest	:Tc2_System.T_MaxString;
END_VAR
getTestNameFor := Tc2_Standard.CONCAT(THIS^.TEST_NAME_PREFIX, nameOfMethodToTest);
END_METHOD

(*

short summary
==================
This test method tests ``assert.dateAndTime.simple.dateAndTime.valueIsEqualTo``
method of CNM_AssertionInterfaces library with various inputs

.. <legal notes>

legal notes
=================
| SPDX-FileCopyrightText: © 2022 ekvip automation GmbH <info@ekvip.de>
| SPDX-License-Identifier: Apache-2.0
| For details check: Apache-2.0_

.. _Apache-2.0: https://www.apache.org/licenses/LICENSE-2.0

.. </legal notes>

*)

METHOD runValueIsEqualToTests
RETURN (NOT TcUnit.TEST_ORDERED(THIS^.getTestNameFor('valueIsEqualTo')));

THIS^.testValueIsEqualTo(
	valueToTest := THIS^.DT_MAX,
	expected := THIS^.DT_MAX
);
THIS^.testValueIsEqualTo(
	valueToTest := THIS^.DT_MIN,
	expected := THIS^.DT_MIN
);
THIS^.testValueIsEqualTo(
	valueToTest := THIS^.DT_MIN,
	expected := THIS^.DT_MAX
);
THIS^.testValueIsEqualTo(
	valueToTest := THIS^.DT_MAX,
	expected := THIS^.DT_MIN
);
THIS^.testValueIsEqualTo(
	valueToTest := THIS^.DT_ALL_NIBBLE_LSB,
	expected := THIS^.DT_ALL_NIBBLE_LSB
);
THIS^.testValueIsEqualTo(
	valueToTest := THIS^.DT_LSB_ONLY,
	expected := THIS^.DT_MSB_ONLY
);
THIS^.testValueIsEqualTo(
	valueToTest := THIS^.DT_MSB_ONLY,
	expected := THIS^.DT_MSB_ONLY
);
THIS^.testValueIsEqualTo(
	valueToTest := THIS^.DT_MSB_ONLY,
	expected := THIS^.DT_LSB_ONLY
);

TcUnit.TEST_FINISHED();
END_METHOD

(*

short summary
==================
This test method tests ``assert.dateAndTime.simple.dateAndTime.valueIsGreaterThan``
method of CNM_AssertionInterfaces library with various inputs

.. <legal notes>

legal notes
=================
| SPDX-FileCopyrightText: © 2022 ekvip automation GmbH <info@ekvip.de>
| SPDX-License-Identifier: Apache-2.0
| For details check: Apache-2.0_

.. _Apache-2.0: https://www.apache.org/licenses/LICENSE-2.0

.. </legal notes>

*)

METHOD runValueIsGreaterThanTests
RETURN (NOT TcUnit.TEST_ORDERED(THIS^.getTestNameFor('valueIsGreaterThan')));

THIS^.testValueIsGreaterThan(
	valueToTest := THIS^.DT_MAX,
	lessValue := THIS^.DT_MAX
);
THIS^.testValueIsGreaterThan(
	valueToTest := THIS^.DT_MIN,
	lessValue := THIS^.DT_MIN
);
THIS^.testValueIsGreaterThan(
	valueToTest := THIS^.DT_MIN,
	lessValue := THIS^.DT_MAX
);
THIS^.testValueIsGreaterThan(
	valueToTest := THIS^.DT_MAX,
	lessValue := THIS^.DT_MIN
);
THIS^.testValueIsGreaterThan(
	valueToTest := THIS^.DT_ALL_NIBBLE_LSB,
	lessValue := THIS^.DT_ALL_NIBBLE_LSB
);
THIS^.testValueIsGreaterThan(
	valueToTest := THIS^.DT_ALL_NIBBLE_MSB,
	lessValue := THIS^.DT_ALL_NIBBLE_LSB
);
THIS^.testValueIsGreaterThan(
	valueToTest := THIS^.DT_ALL_NIBBLE_LSB,
	lessValue := THIS^.DT_ALL_NIBBLE_MSB
);
THIS^.testValueIsGreaterThan(
	valueToTest := THIS^.DT_LSB_ONLY,
	lessValue := THIS^.DT_MSB_ONLY
);
THIS^.testValueIsGreaterThan(
	valueToTest := THIS^.DT_MSB_ONLY,
	lessValue := THIS^.DT_MSB_ONLY
);
THIS^.testValueIsGreaterThan(
	valueToTest := THIS^.DT_MSB_ONLY,
	lessValue := THIS^.DT_LSB_ONLY
);
THIS^.testValueIsGreaterThan(
	valueToTest := THIS^.DT_LSB_IS_UNSET,
	lessValue := THIS^.DT_MAX
);
THIS^.testValueIsGreaterThan(
	valueToTest := THIS^.DT_MAX,
	lessValue := THIS^.DT_LSB_IS_UNSET
);
TcUnit.TEST_FINISHED();
END_METHOD

(*

short summary
==================
This test method tests ``assert.dateAndTime.simple.dateAndTime.valueIsInRangeOf``
method of CNM_AssertionInterfaces library with various inputs

.. <legal notes>

legal notes
=================
| SPDX-FileCopyrightText: © 2022 ekvip automation GmbH <info@ekvip.de>
| SPDX-License-Identifier: Apache-2.0
| For details check: Apache-2.0_

.. _Apache-2.0: https://www.apache.org/licenses/LICENSE-2.0

.. </legal notes>

*)

METHOD runValueIsInRangeOfTests
RETURN (NOT TcUnit.TEST_ORDERED(THIS^.getTestNameFor('valueIsInRangeOf')));

THIS^.testValueIsInRangeOf(
	lowerLimit := THIS^.DT_MIN,
	valueToTest := THIS^.DT_MAX,
	upperLimit	:= THIS^.DT_MAX
);
THIS^.testValueIsInRangeOf(
	lowerLimit := THIS^.DT_MIN,
	valueToTest := THIS^.DT_MIN,
	upperLimit	:= THIS^.DT_MAX
);
THIS^.testValueIsInRangeOf(
	lowerLimit := THIS^.DT_MAX,
	valueToTest := THIS^.DT_MAX,
	upperLimit	:= THIS^.DT_MIN
);
THIS^.testValueIsInRangeOf(
	lowerLimit := THIS^.DT_MAX,
	valueToTest := THIS^.DT_MIN,
	upperLimit	:= THIS^.DT_MIN
);
THIS^.testValueIsInRangeOf(
	lowerLimit := THIS^.DT_LSB_IS_UNSET,
	valueToTest := THIS^.DT_MIN,
	upperLimit	:= THIS^.DT_MAX
);
THIS^.testValueIsInRangeOf(
	lowerLimit := THIS^.DT_MIN,
	valueToTest := THIS^.DT_LSB_IS_UNSET,
	upperLimit	:= THIS^.DT_MAX
);
THIS^.testValueIsInRangeOf(
	lowerLimit := THIS^.DT_LSB_IS_UNSET,
	valueToTest := THIS^.DT_LSB_IS_UNSET,
	upperLimit	:= THIS^.DT_LSB_IS_UNSET
);
THIS^.testValueIsInRangeOf(
	lowerLimit := THIS^.DT_ALL_NIBBLE_LSB,
	valueToTest := THIS^.DT_LSB_IS_UNSET,
	upperLimit	:= THIS^.DT_ALL_NIBBLE_MSB
);
THIS^.testValueIsInRangeOf(
	lowerLimit := THIS^.DT_LSB_IS_UNSET,
	valueToTest := THIS^.DT_ALL_NIBBLE_LSB,
	upperLimit	:= THIS^.DT_ALL_NIBBLE_MSB
);
THIS^.testValueIsInRangeOf(
	lowerLimit := THIS^.DT_LSB_ONLY,
	valueToTest := THIS^.DT_WITHOUT_MSB,
	upperLimit	:= THIS^.DT_MSB_ONLY
);
THIS^.testValueIsInRangeOf(
	lowerLimit := THIS^.DT_WITHOUT_MSB,
	valueToTest := THIS^.DT_LSB_ONLY,
	upperLimit	:= THIS^.DT_MSB_ONLY
);
THIS^.testValueIsInRangeOf(
	lowerLimit := THIS^.DT_WITHOUT_NIBBLE_MSB,
	valueToTest := THIS^.DT_MAX,
	upperLimit	:= THIS^.DT_ALL_NIBBLE_MSB
);
THIS^.testValueIsInRangeOf(
	lowerLimit := THIS^.DT_WITHOUT_NIBBLE_MSB,
	valueToTest := THIS^.DT_MIN,
	upperLimit	:= THIS^.DT_ALL_NIBBLE_MSB
);
THIS^.testValueIsInRangeOf(
	lowerLimit := THIS^.DT_WITHOUT_NIBBLE_MSB,
	valueToTest := THIS^.DT_WITHOUT_NIBBLE_MSB,
	upperLimit	:= THIS^.DT_ALL_NIBBLE_MSB
);
THIS^.testValueIsInRangeOf(
	lowerLimit := THIS^.DT_WITHOUT_NIBBLE_MSB,
	valueToTest := THIS^.DT_ALL_NIBBLE_MSB,
	upperLimit	:= THIS^.DT_ALL_NIBBLE_MSB
);
TcUnit.TEST_FINISHED();
END_METHOD

(*

short summary
==================
This test method tests ``assert.dateAndTime.simple.dateAndTime.valueIsLessThan``
method of CNM_AssertionInterfaces library with various inputs

.. <legal notes>

legal notes
=================
| SPDX-FileCopyrightText: © 2022 ekvip automation GmbH <info@ekvip.de>
| SPDX-License-Identifier: Apache-2.0
| For details check: Apache-2.0_

.. _Apache-2.0: https://www.apache.org/licenses/LICENSE-2.0

.. </legal notes>

*)

METHOD runValueIsLessThanTests
RETURN (NOT TcUnit.TEST_ORDERED(THIS^.getTestNameFor('valueIsLessThan')));

THIS^.testValueIsLessThan(
	valueToTest := THIS^.DT_MAX,
	greaterValue := THIS^.DT_MAX
);
THIS^.testValueIsLessThan(
	valueToTest := THIS^.DT_MIN,
	greaterValue := THIS^.DT_MIN
);
THIS^.testValueIsLessThan(
	valueToTest := THIS^.DT_MIN,
	greaterValue := THIS^.DT_MAX
);
THIS^.testValueIsLessThan(
	valueToTest := THIS^.DT_MAX,
	greaterValue := THIS^.DT_MIN
);
THIS^.testValueIsLessThan(
	valueToTest := THIS^.DT_ALL_NIBBLE_LSB,
	greaterValue := THIS^.DT_ALL_NIBBLE_LSB
);
THIS^.testValueIsLessThan(
	valueToTest := THIS^.DT_ALL_NIBBLE_MSB,
	greaterValue := THIS^.DT_ALL_NIBBLE_LSB
);
THIS^.testValueIsLessThan(
	valueToTest := THIS^.DT_ALL_NIBBLE_LSB,
	greaterValue := THIS^.DT_ALL_NIBBLE_MSB
);
THIS^.testValueIsLessThan(
	valueToTest := THIS^.DT_LSB_ONLY,
	greaterValue := THIS^.DT_MSB_ONLY
);
THIS^.testValueIsLessThan(
	valueToTest := THIS^.DT_MSB_ONLY,
	greaterValue := THIS^.DT_MSB_ONLY
);
THIS^.testValueIsLessThan(
	valueToTest := THIS^.DT_MSB_ONLY,
	greaterValue := THIS^.DT_LSB_ONLY
);
THIS^.testValueIsLessThan(
	valueToTest := THIS^.DT_LSB_IS_UNSET,
	greaterValue := THIS^.DT_MAX
);
THIS^.testValueIsLessThan(
	valueToTest := THIS^.DT_MAX,
	greaterValue := THIS^.DT_LSB_IS_UNSET
);
TcUnit.TEST_FINISHED();
END_METHOD

(*

short summary
==================
This test method tests ``assert.dateAndTime.simple.dateAndTime.valueIsMax``
method of CNM_AssertionInterfaces library with various inputs

.. <legal notes>

legal notes
=================
| SPDX-FileCopyrightText: © 2022 ekvip automation GmbH <info@ekvip.de>
| SPDX-License-Identifier: Apache-2.0
| For details check: Apache-2.0_

.. _Apache-2.0: https://www.apache.org/licenses/LICENSE-2.0

.. </legal notes>

*)

METHOD runValueIsMaxTests
RETURN (NOT TcUnit.TEST_ORDERED(THIS^.getTestNameFor('valueIsMax')));

THIS^.testValueIsMax(
	valueToTest := THIS^.DT_MAX,
	maximumValue := THIS^.DT_MAX
);
THIS^.testValueIsMax(
	valueToTest := THIS^.DT_MIN,
	maximumValue := THIS^.DT_MIN
);
THIS^.testValueIsMax(
	valueToTest := THIS^.DT_MIN,
	maximumValue := THIS^.DT_MAX
);
THIS^.testValueIsMax(
	valueToTest := THIS^.DT_MAX,
	maximumValue := THIS^.DT_MIN
);
THIS^.testValueIsMax(
	valueToTest := THIS^.DT_ALL_NIBBLE_LSB,
	maximumValue := THIS^.DT_ALL_NIBBLE_LSB
);
THIS^.testValueIsMax(
	valueToTest := THIS^.DT_ALL_NIBBLE_MSB,
	maximumValue := THIS^.DT_ALL_NIBBLE_LSB
);
THIS^.testValueIsMax(
	valueToTest := THIS^.DT_ALL_NIBBLE_LSB,
	maximumValue := THIS^.DT_ALL_NIBBLE_MSB
);
THIS^.testValueIsMax(
	valueToTest := THIS^.DT_LSB_ONLY,
	maximumValue := THIS^.DT_MSB_ONLY
);
THIS^.testValueIsMax(
	valueToTest := THIS^.DT_MSB_ONLY,
	maximumValue := THIS^.DT_MSB_ONLY
);
THIS^.testValueIsMax(
	valueToTest := THIS^.DT_MSB_ONLY,
	maximumValue := THIS^.DT_LSB_ONLY
);
THIS^.testValueIsMax(
	valueToTest := THIS^.DT_LSB_IS_UNSET,
	maximumValue := THIS^.DT_MAX
);
THIS^.testValueIsMax(
	valueToTest := THIS^.DT_MAX,
	maximumValue := THIS^.DT_LSB_IS_UNSET
);
TcUnit.TEST_FINISHED();
END_METHOD

(*

short summary
==================
This test method tests ``assert.dateAndTime.simple.dateAndTime.valueIsMin``
method of CNM_AssertionInterfaces library with various inputs

.. <legal notes>

legal notes
=================
| SPDX-FileCopyrightText: © 2022 ekvip automation GmbH <info@ekvip.de>
| SPDX-License-Identifier: Apache-2.0
| For details check: Apache-2.0_

.. _Apache-2.0: https://www.apache.org/licenses/LICENSE-2.0

.. </legal notes>

*)

METHOD runValueIsMinTests
RETURN (NOT TcUnit.TEST_ORDERED(THIS^.getTestNameFor('valueIsMin')));

THIS^.testValueIsMin(
	valueToTest := THIS^.DT_MAX,
	minimumValue := THIS^.DT_MAX
);
THIS^.testValueIsMin(
	valueToTest := THIS^.DT_MIN,
	minimumValue := THIS^.DT_MIN
);
THIS^.testValueIsMin(
	valueToTest := THIS^.DT_MIN,
	minimumValue := THIS^.DT_MAX
);
THIS^.testValueIsMin(
	valueToTest := THIS^.DT_MAX,
	minimumValue := THIS^.DT_MIN
);
THIS^.testValueIsMin(
	valueToTest := THIS^.DT_ALL_NIBBLE_LSB,
	minimumValue := THIS^.DT_ALL_NIBBLE_LSB
);
THIS^.testValueIsMin(
	valueToTest := THIS^.DT_ALL_NIBBLE_MSB,
	minimumValue := THIS^.DT_ALL_NIBBLE_LSB
);
THIS^.testValueIsMin(
	valueToTest := THIS^.DT_ALL_NIBBLE_LSB,
	minimumValue := THIS^.DT_ALL_NIBBLE_MSB
);
THIS^.testValueIsMin(
	valueToTest := THIS^.DT_LSB_ONLY,
	minimumValue := THIS^.DT_MSB_ONLY
);
THIS^.testValueIsMin(
	valueToTest := THIS^.DT_MSB_ONLY,
	minimumValue := THIS^.DT_MSB_ONLY
);
THIS^.testValueIsMin(
	valueToTest := THIS^.DT_MSB_ONLY,
	minimumValue := THIS^.DT_LSB_ONLY
);
THIS^.testValueIsMin(
	valueToTest := THIS^.DT_LSB_IS_UNSET,
	minimumValue := THIS^.DT_MAX
);
THIS^.testValueIsMin(
	valueToTest := THIS^.DT_MAX,
	minimumValue := THIS^.DT_LSB_IS_UNSET
);
TcUnit.TEST_FINISHED();
END_METHOD

(*

short summary
==================
This test method tests ``assert.dateAndTime.simple.dateAndTime.valueIsNotEqualTo``
method of CNM_AssertionInterfaces library with various inputs

.. <legal notes>

legal notes
=================
| SPDX-FileCopyrightText: © 2022 ekvip automation GmbH <info@ekvip.de>
| SPDX-License-Identifier: Apache-2.0
| For details check: Apache-2.0_

.. _Apache-2.0: https://www.apache.org/licenses/LICENSE-2.0

.. </legal notes>

*)

METHOD runValueIsNotEqualToTests
RETURN (NOT TcUnit.TEST_ORDERED(THIS^.getTestNameFor('valueIsNotEqualTo')));

THIS^.testValueIsNotEqualTo(
	valueToTest := THIS^.DT_MAX,
	unexpectedValue := THIS^.DT_MAX
);
THIS^.testValueIsNotEqualTo(
	valueToTest := THIS^.DT_MIN,
	unexpectedValue := THIS^.DT_MIN
);
THIS^.testValueIsNotEqualTo(
	valueToTest := THIS^.DT_MIN,
	unexpectedValue := THIS^.DT_MAX
);
THIS^.testValueIsNotEqualTo(
	valueToTest := THIS^.DT_MAX,
	unexpectedValue := THIS^.DT_MIN
);
THIS^.testValueIsNotEqualTo(
	valueToTest := THIS^.DT_ALL_NIBBLE_LSB,
	unexpectedValue := THIS^.DT_ALL_NIBBLE_LSB
);
THIS^.testValueIsNotEqualTo(
	valueToTest := THIS^.DT_LSB_ONLY,
	unexpectedValue := THIS^.DT_MSB_ONLY
);
THIS^.testValueIsNotEqualTo(
	valueToTest := THIS^.DT_MSB_ONLY,
	unexpectedValue := THIS^.DT_MSB_ONLY
);
THIS^.testValueIsNotEqualTo(
	valueToTest := THIS^.DT_MSB_ONLY,
	unexpectedValue := THIS^.DT_LSB_ONLY
);

TcUnit.TEST_FINISHED();
END_METHOD

(*

short summary
==================
This test method tests ``assert.dateAndTime.simple.dateAndTime.valueIsEqualTo``
method of CNM_AssertionInterfaces library, 
it provides the possibility to handover test data via parameter 


.. <legal notes>

legal notes
=================
| SPDX-FileCopyrightText: © 2022 ekvip automation GmbH <info@ekvip.de>
| SPDX-License-Identifier: Apache-2.0
| For details check: Apache-2.0_

.. _Apache-2.0: https://www.apache.org/licenses/LICENSE-2.0

.. </legal notes>

parameters
==========

*)

METHOD testValueIsEqualTo 
VAR_INPUT
	(* for the test it's the parameter ``currentValue`` *)
	valueToTest	:DT;
	(* for the test it's the parameter ``expectedValue`` *)
	expected	:DT;
END_VAR
VAR
	(* just the expectation if the assertion to test must be worng or true *)
	assertionIsWrong		:BOOL;
	(* contains the format string for the test message *)
	message					:Tc2_System.T_MaxString;
	(* TwinCAT printf with the test message *)
	messageStringBuilder	:Tc2_Utilities.FB_FormatString;
	(* dt value of ``currentValue`` as string *)
	currentValueAsString	:STRING(22);
	(* dt value of ``expectedValue`` as string *)
	expectedValueAsString	:STRING(22);
END_VAR
THIS^.assertorContainer.resetAssertor();

assertionIsWrong := (valueToTest <> expected);
message := SEL(
	assertionIsWrong,
	'currentValue is %s expectedValue is %s assertion must be TRUE', 
	'currentValue is %s expectedValue is %s assertion must be FALSE'
);
currentValueAsString := TO_STRING(valueToTest);
expectedValueAsString := TO_STRING(expected);

messageStringBuilder(
	sFormat := message,
	arg1 := THIS^.AnyToArg(currentValueAsString),
	arg2 := THIS^.AnyToArg(expectedValueAsString)
);

THIS^.assertorContainer.assertor.assert.dateAndTime.simple.dateAndTime.valueIsEqualTo(
	currentValue	:= valueToTest,
	expectedValue	:= expected,
	message			:= ''
);

THIS^.AssertEquals_BOOL(
	Expected 	:= assertionIsWrong,
	Actual 		:= THIS^.assertorContainer.wasAssertionWrong,
	Message 	:= messageStringBuilder.sOut
);
END_METHOD

(*

short summary
==================
This test method tests ``assert.dateAndTime.simple.dateAndTime.valueIsGreaterThan``
method of CNM_AssertionInterfaces library, 
it provides the possibility to handover test data via parameter 


.. <legal notes>

legal notes
=================
| SPDX-FileCopyrightText: © 2022 ekvip automation GmbH <info@ekvip.de>
| SPDX-License-Identifier: Apache-2.0
| For details check: Apache-2.0_

.. _Apache-2.0: https://www.apache.org/licenses/LICENSE-2.0

.. </legal notes>

parameters
==========

*)

METHOD testValueIsGreaterThan 
VAR_INPUT
	(* for the test it's the parameter ``currentValue`` *)
	valueToTest	:DT;
	(* for the test it's the parameter ``lessValue`` *)
	lessValue	:DT;
END_VAR
VAR
	(* just the expectation if the assertion to test must be worng or true *)
	assertionIsWrong		:BOOL;
	(* contains the format string for the test message *)
	message					:Tc2_System.T_MaxString;
	(* TwinCAT printf with the test message *)
	messageStringBuilder	:Tc2_Utilities.FB_FormatString;
	(* dt value of ``currentValue`` as string *)
	currentValueAsString	:STRING(22);
	(* dt value of ``lessValue`` as string *)
	lessValueAsString		:STRING(22);
END_VAR
THIS^.assertorContainer.resetAssertor();

assertionIsWrong := (valueToTest <= lessValue);
message := SEL(
	assertionIsWrong,
	'currentValue is %s lessValue is %s assertion must be TRUE', 
	'currentValue is %s lessValue is %s assertion must be FALSE'
);
currentValueAsString := TO_STRING(valueToTest);
lessValueAsString := TO_STRING(lessValue);

messageStringBuilder(
	sFormat := message,
	arg1 := THIS^.AnyToArg(currentValueAsString),
	arg2 := THIS^.AnyToArg(lessValueAsString)
);

THIS^.assertorContainer.assertor.assert.dateAndTime.simple.dateAndTime.valueIsGreaterThan(
	currentValue	:= valueToTest,
	lessValue		:= lessValue,
	message			:= ''
);

THIS^.AssertEquals_BOOL(
	Expected 	:= assertionIsWrong,
	Actual 		:= THIS^.assertorContainer.wasAssertionWrong,
	Message 	:= messageStringBuilder.sOut
);
END_METHOD

(*

short summary
==================
This test method tests ``assert.dateAndTime.simple.dateAndTime.valueIsInRangeOf``
method of CNM_AssertionInterfaces library, 
it provides the possibility to handover test data via parameter 


.. <legal notes>

legal notes
=================
| SPDX-FileCopyrightText: © 2022 ekvip automation GmbH <info@ekvip.de>
| SPDX-License-Identifier: Apache-2.0
| For details check: Apache-2.0_

.. _Apache-2.0: https://www.apache.org/licenses/LICENSE-2.0

.. </legal notes>

parameters
==========

*)

METHOD testValueIsInRangeOf 
VAR_INPUT
	(* for the test it's the parameter ``lowerLimit`` *)
	lowerLimit	:DT;
	(* for the test it's the parameter ``currentValue`` *)
	valueToTest	:DT;
	(* for the test it's the parameter ``upperLimit`` *)
	upperLimit	:DT;
END_VAR
VAR
	(* just the expectation if the assertion to test must be worng or true *)
	assertionIsWrong		:BOOL;
	(* contains the format string for the test message *)
	message					:Tc2_System.T_MaxString;
	(* TwinCAT printf with the test message *)
	messageStringBuilder	:Tc2_Utilities.FB_FormatString;
	(* dt value of ``lowerLimit`` as string *)
	lowerLimitAsString		:STRING(22);
	(* dt value of ``currentValue`` as string *)
	currentValueAsString	:STRING(22);
	(* dt value of ``upperLimit`` as string *)
	upperLimitAsString		:STRING(22);

END_VAR
THIS^.assertorContainer.resetAssertor();

assertionIsWrong := ((valueToTest < lowerLimit) OR (valueToTest > upperLimit));
message := SEL(
	assertionIsWrong,
	'lowerLimit is %s currentValue is %s upperLimit is %s assertion must be TRUE', 
	'lowerLimit is %s currentValue is %s upperLimit is %s assertion must be FALSE'
);
lowerLimitAsString		:= TO_STRING(lowerLimit);
currentValueAsString	:= TO_STRING(valueToTest);
upperLimitAsString		:= TO_STRING(upperLimit);

messageStringBuilder(
	sFormat := message,
	arg1 := THIS^.AnyToArg(lowerLimitAsString),
	arg2 := THIS^.AnyToArg(currentValueAsString),
	arg3 := THIS^.AnyToArg(upperLimitAsString)
);

THIS^.assertorContainer.assertor.assert.dateAndTime.simple.dateAndTime.valueIsInRangeOf(
	lowerLimit		:= lowerLimit,
	currentValue	:= valueToTest,
	upperLimit		:= upperLimit,
	message			:= ''
);

THIS^.AssertEquals_BOOL(
	Expected 	:= assertionIsWrong,
	Actual 		:= THIS^.assertorContainer.wasAssertionWrong,
	Message 	:= messageStringBuilder.sOut
);
END_METHOD

(*

short summary
==================
This test method tests ``assert.dateAndTime.simple.dateAndTime.valueIsLessThan``
method of CNM_AssertionInterfaces library, 
it provides the possibility to handover test data via parameter 


.. <legal notes>

legal notes
=================
| SPDX-FileCopyrightText: © 2022 ekvip automation GmbH <info@ekvip.de>
| SPDX-License-Identifier: Apache-2.0
| For details check: Apache-2.0_

.. _Apache-2.0: https://www.apache.org/licenses/LICENSE-2.0

.. </legal notes>

parameters
==========

*)

METHOD testValueIsLessThan 
VAR_INPUT
	(* for the test it's the parameter ``currentValue`` *)
	valueToTest		:DT;
	(* for the test it's the parameter ``greaterValue`` *)
	greaterValue	:DT;
END_VAR
VAR
	(* just the expectation if the assertion to test must be worng or true *)
	assertionIsWrong		:BOOL;
	(* contains the format string for the test message *)
	message					:Tc2_System.T_MaxString;
	(* TwinCAT printf with the test message *)
	messageStringBuilder	:Tc2_Utilities.FB_FormatString;
	(* dt value of ``currentValue`` as string *)
	currentValueAsString	:STRING(22);
	(* dt value of ``greaterValue`` as string *)
	greaterValueAsString	:STRING(22);
END_VAR
THIS^.assertorContainer.resetAssertor();

assertionIsWrong := (valueToTest >= greaterValue);
message := SEL(
	assertionIsWrong,
	'currentValue is %s greaterValue is %s assertion must be TRUE', 
	'currentValue is %s greaterValue is %s assertion must be FALSE'
);
currentValueAsString := TO_STRING(valueToTest);
greaterValueAsString := TO_STRING(greaterValue);

messageStringBuilder(
	sFormat := message,
	arg1 := THIS^.AnyToArg(currentValueAsString),
	arg2 := THIS^.AnyToArg(greaterValueAsString)
);

THIS^.assertorContainer.assertor.assert.dateAndTime.simple.dateAndTime.valueIsLessThan(
	currentValue	:= valueToTest,
	greaterValue	:= greaterValue,
	message			:= ''
);

THIS^.AssertEquals_BOOL(
	Expected 	:= assertionIsWrong,
	Actual 		:= THIS^.assertorContainer.wasAssertionWrong,
	Message 	:= messageStringBuilder.sOut
);
END_METHOD

(*

short summary
==================
This test method tests ``assert.dateAndTime.simple.dateAndTime.valueIsMax``
method of CNM_AssertionInterfaces library, 
it provides the possibility to handover test data via parameter 


.. <legal notes>

legal notes
=================
| SPDX-FileCopyrightText: © 2022 ekvip automation GmbH <info@ekvip.de>
| SPDX-License-Identifier: Apache-2.0
| For details check: Apache-2.0_

.. _Apache-2.0: https://www.apache.org/licenses/LICENSE-2.0

.. </legal notes>

parameters
==========

*)

METHOD testValueIsMax 
VAR_INPUT
	(* for the test it's the parameter ``currentValue`` *)
	valueToTest		:DT;
	(* for the test it's the parameter ``greaterValue`` *)
	maximumValue	:DT;
END_VAR
VAR
	(* just the expectation if the assertion to test must be worng or true *)
	assertionIsWrong		:BOOL;
	(* contains the format string for the test message *)
	message					:Tc2_System.T_MaxString;
	(* TwinCAT printf with the test message *)
	messageStringBuilder	:Tc2_Utilities.FB_FormatString;
	(* dt value of ``currentValue`` as string *)
	currentValueAsString	:STRING(22);
	(* dt value of ``maximumValue`` as string *)
	maximumValueAsString	:STRING(22);
END_VAR
THIS^.assertorContainer.resetAssertor();

assertionIsWrong := (valueToTest > maximumValue);
message := SEL(
	assertionIsWrong,
	'currentValue is %s maximumValue is %s assertion must be TRUE', 
	'currentValue is %s maximumValue is %s assertion must be FALSE'
);
currentValueAsString := TO_STRING(valueToTest);
maximumValueAsString := TO_STRING(maximumValue);

messageStringBuilder(
	sFormat := message,
	arg1 := THIS^.AnyToArg(currentValueAsString),
	arg2 := THIS^.AnyToArg(maximumValueAsString)
);

THIS^.assertorContainer.assertor.assert.dateAndTime.simple.dateAndTime.valueIsMax(
	currentValue	:= valueToTest,
	maximumValue	:= maximumValue,
	message			:= ''
);

THIS^.AssertEquals_BOOL(
	Expected 	:= assertionIsWrong,
	Actual 		:= THIS^.assertorContainer.wasAssertionWrong,
	Message 	:= messageStringBuilder.sOut
);
END_METHOD

(*

short summary
==================
This test method tests ``assert.dateAndTime.simple.dateAndTime.valueIsMin``
method of CNM_AssertionInterfaces library, 
it provides the possibility to handover test data via parameter 


.. <legal notes>

legal notes
=================
| SPDX-FileCopyrightText: © 2022 ekvip automation GmbH <info@ekvip.de>
| SPDX-License-Identifier: Apache-2.0
| For details check: Apache-2.0_

.. _Apache-2.0: https://www.apache.org/licenses/LICENSE-2.0

.. </legal notes>

parameters
==========

*)

METHOD testValueIsMin 
VAR_INPUT
	(* for the test it's the parameter ``currentValue`` *)
	valueToTest		:DT;
	(* for the test it's the parameter ``greaterValue`` *)
	minimumValue	:DT;
END_VAR
VAR
	(* just the expectation if the assertion to test must be worng or true *)
	assertionIsWrong		:BOOL;
	(* contains the format string for the test message *)
	message					:Tc2_System.T_MaxString;
	(* TwinCAT printf with the test message *)
	messageStringBuilder	:Tc2_Utilities.FB_FormatString;
	(* dt value of ``currentValue`` as string *)
	currentValueAsString	:STRING(22);
	(* dt value of ``minimumValue`` as string *)
	minimumValueAsString	:STRING(22);
END_VAR
THIS^.assertorContainer.resetAssertor();

assertionIsWrong := (valueToTest < minimumValue);
message := SEL(
	assertionIsWrong,
	'currentValue is %s minimumValue is %s assertion must be TRUE', 
	'currentValue is %s minimumValue is %s assertion must be FALSE'
);
currentValueAsString := TO_STRING(valueToTest);
minimumValueAsString := TO_STRING(minimumValue);

